  MoveL 1910 to (-109.13, -104.27, -4.96) mm, rotated rx 88.64 ry 0 rz 132.9 deg; joints [121.787, -25.073, 45.669, -119.581, 37.28, 191.868, 25, -132.901]
  MoveL 1911 to (-113.05, -99.53, -11.02) mm, rotated rx 86.5 ry 0 rz 130.7 deg; joints [121.42, -25.047, 46.567, -120.984, 37.45, 195.607, 25, -130.697]
  MoveL 1912 to (-113.34, -99.15, -11.43) mm, rotated rx 86.38 ry 0 rz 130.56 deg; joints [121.402, -25.048, 46.621, -121.062, 37.463, 195.813, 25, -130.561]
  MoveL 1913 to (-115.31, -96.51, -13.99) mm, rotated rx 85.43 ry 0 rz 129.34 deg; joints [121.25, -25.013, 47.005, -121.68, 37.561, 197.469, 25, -129.342]
  MoveL 1914 to (-115.68, -96.01, -14.39) mm, rotated rx 85.34 ry 0 rz 129.19 deg; joints [121.239, -25.019, 47.054, -121.738, 37.575, 197.627, 25, -129.193]
  MoveL 1915 to (-118.09, -92.7, -16.37) mm, rotated rx 84.63 ry 0 rz 127.72 deg; joints [121.132, -24.991, 47.345, -122.198, 37.66, 198.867, 25, -127.716]
  MoveL 1916 to (-118.46, -92.16, -16.77) mm, rotated rx 84.44 ry 0 rz 127.39 deg; joints [121.1, -24.97, 47.412, -122.327, 37.681, 199.21, 25, -127.39]
  MoveL 1917 to (-121.85, -86.42, -22.18) mm, rotated rx 82.29 ry 0 rz 124.74 deg; joints [120.788, -24.794, 48.227, -123.721, 37.981, 202.967, 25, -124.738]
  MoveL 1918 to (-122.46, -84.98, -24.25) mm, rotated rx 81.33 ry 0 rz 123.99 deg; joints [120.657, -24.684, 48.564, -124.332, 38.131, 204.635, 25, -123.992]
  MoveL 1919 to (-122.65, -84.59, -24.68) mm, rotated rx 81.33 ry 0 rz 123.99 deg; joints [120.661, -24.702, 48.591, -124.337, 38.14, 204.644, 25, -123.992]
  MoveL 1920 to (-122.81, -84.27, -24.97) mm, rotated rx 81.22 ry 0 rz 123.85 deg; joints [120.647, -24.69, 48.632, -124.407, 38.159, 204.837, 25, -123.853]
  MoveL 1921 to (-124.4, -81.2, -27.15) mm, rotated rx 80.44 ry 0 rz 122.62 deg; joints [120.554, -24.613, 48.934, -124.902, 38.304, 206.195, 25, -122.615]
  MoveL 1922 to (-124.78, -79.6, -30.03) mm, rotated rx 78.99 ry 0 rz 121.69 deg; joints [120.374, -24.397, 49.413, -125.811, 38.573, 208.715, 25, -121.69]
  MoveL 1923 to (-124.89, -79.17, -30.67) mm, rotated rx 78.81 ry 0 rz 121.57 deg; joints [120.355, -24.376, 49.486, -125.927, 38.614, 209.031, 25, -121.568]
  MoveL 1924 to (-125.14, -77.59, -33.5) mm, rotated rx 77.62 ry 0 rz 120.94 deg; joints [120.228, -24.195, 49.899, -126.663, 38.874, 211.098, 25, -120.935]
  MoveL 1925 to (-125.14, -77.57, -33.6) mm, rotated rx 76.62 ry 0 rz 120.98 deg; joints [120.153, -24.074, 50.182, -127.145, 39.063, 212.676, 25, -120.981]
  MoveL 1926 to (-124.65, -77.98, -34.49) mm, rotated rx 76.27 ry 0 rz 121.22 deg; joints [120.121, -24.015, 50.302, -127.356, 39.148, 213.273, 25, -121.217]
  MoveL 1927 to (-124.35, -78.16, -35.13) mm, rotated rx 76.27 ry 0 rz 121.22 deg; joints [120.109, -23.99, 50.31, -127.401, 39.159, 213.325, 25, -121.217]
  MoveL 1928 to (-124.19, -78.22, -35.56) mm, rotated rx 76.11 ry 0 rz 121.27 deg; joints [120.094, -23.961, 50.368, -127.503, 39.201, 213.615, 25, -121.269]
  MoveL 1929 to (-123.95, -78.19, -36.45) mm, rotated rx 76.11 ry 0 rz 121.27 deg; joints [120.085, -23.943, 50.39, -127.552, 39.22, 213.673, 25, -121.269]
  MoveL 1930 to (-123.38, -77.54, -39.6) mm, rotated rx 74.87 ry 0 rz 121.17 deg; joints [119.981, -23.712, 50.808, -128.292, 39.545, 215.805, 25, -121.168]
  MoveL 1931 to (-120.74, -79.41, -43.84) mm, rotated rx 72.6 ry 0 rz 122.5 deg; joints [119.836, -23.279, 51.521, -129.525, 40.165, 219.593, 25, -122.503]
  MoveL 1932 to (-120.21, -79.55, -45.03) mm, rotated rx 72.6 ry 0 rz 122.5 deg; joints [119.821, -23.236, 51.54, -129.599, 40.194, 219.681, 25, -122.503]
  MoveL 1933 to (-119.97, -79.45, -45.84) mm, rotated rx 72.28 ry 0 rz 122.52 deg; joints [119.801, -23.161, 51.642, -129.781, 40.294, 220.231, 25, -122.52]
  MoveL 1934 to (-117.99, -78.14, -52.73) mm, rotated rx 69.57 ry 0 rz 122.5 deg; joints [119.669, -22.465, 52.47, -131.278, 41.197, 224.832, 25, -122.503]
  MoveL 1935 to (-116.68, -77.5, -56.45) mm, rotated rx 68.02 ry 0 rz 122.57 deg; joints [119.621, -22.022, 52.911, -132.08, 41.754, 227.415, 25, -122.572]
  MoveL 1936 to (-116.44, -76.93, -57.7) mm, rotated rx 68.02 ry 0 rz 122.57 deg; joints [119.626, -22.007, 52.954, -132.122, 41.795, 227.475, 25, -122.572]
  MoveL 1937 to (-116.45, -76.65, -58.07) mm, rotated rx 67.87 ry 0 rz 122.47 deg; joints [119.622, -21.962, 52.996, -132.199, 41.852, 227.727, 25, -122.474]
  MoveL 1938 to (-116.52, -76.14, -58.6) mm, rotated rx 67.87 ry 0 rz 122.47 deg; joints [119.631, -21.972, 53.025, -132.204, 41.871, 227.74, 25, -122.474]
  MoveL 1939 to (-117.45, -71.82, -62.09) mm, rotated rx 66.42 ry 0 rz 120.74 deg; joints [119.607, -21.514, 53.417, -132.923, 42.43, 230.138, 25, -120.743]
  MoveL 1940 to (-117.61, -71.24, -62.45) mm, rotated rx 66.42 ry 0 rz 120.74 deg; joints [119.62, -21.534, 53.445, -132.916, 42.444, 230.138, 25, -120.743]
  MoveL 1941 to (-117.78, -70.77, -62.67) mm, rotated rx 66.33 ry 0 rz 120.54 deg; joints [119.619, -21.504, 53.469, -132.96, 42.48, 230.287, 25, -120.541]
  MoveL 1942 to (-119.62, -65.95, -64.4) mm, rotated rx 65.65 ry 0 rz 118.51 deg; joints [119.619, -21.283, 53.659, -133.285, 42.761, 231.416, 25, -118.506]
  MoveL 1943 to (-119.93, -63.2, -66.55) mm, rotated rx 64.56 ry 0 rz 117.09 deg; joints [119.603, -20.877, 53.896, -133.804, 43.193, 233.202, 25, -117.086]
  MoveL 1944 to (-120.07, -62.36, -67.09) mm, rotated rx 64.4 ry 0 rz 116.84 deg; joints [119.609, -20.828, 53.946, -133.874, 43.266, 233.458, 25, -116.837]
  MoveL 1945 to (-120.27, -59.5, -69.25) mm, rotated rx 63.41 ry 0 rz 115.6 deg; joints [119.614, -20.455, 54.174, -134.322, 43.687, 235.077, 25, -115.604]
  MoveL 1946 to (-120.29, -59.56, -69.2) mm, rotated rx 62.39 ry 0 rz 115.34 deg; joints [119.613, -20.12, 54.335, -134.692, 44.035, 236.603, 25, -115.342]
  MoveL 1947 to (-119.61, -59.72, -70.24) mm, rotated rx 61.95 ry 0 rz 115.53 deg; joints [119.623, -19.948, 54.435, -134.879, 44.231, 237.311, 25, -115.527]
  MoveL 1948 to (-119.15, -59.77, -70.98) mm, rotated rx 61.71 ry 0 rz 115.61 deg; joints [119.628, -19.842, 54.491, -134.99, 44.349, 237.717, 25, -115.606]
  MoveL 1949 to (-118.82, -59.72, -71.58) mm, rotated rx 61.71 ry 0 rz 115.61 deg; joints [119.628, -19.815, 54.5, -135.017, 44.374, 237.754, 25, -115.606]
  MoveL 1950 to (-115.87, -58.28, -77.36) mm, rotated rx 59.18 ry 0 rz 115.6 deg; joints [119.722, -18.764, 55.025, -136.014, 45.553, 241.762, 25, -115.596]
  MoveL 1951 to (-115.4, -57.54, -78.6) mm, rotated rx 59.18 ry 0 rz 115.6 deg; joints [119.738, -18.736, 55.064, -136.041, 45.61, 241.814, 25, -115.596]
  MoveL 1952 to (-115.3, -56.99, -79.15) mm, rotated rx 58.94 ry 0 rz 115.39 deg; joints [119.75, -18.628, 55.111, -136.132, 45.728, 242.2, 25, -115.393]
  MoveL 1953 to (-115.31, -56.09, -79.78) mm, rotated rx 58.94 ry 0 rz 115.39 deg; joints [119.771, -18.644, 55.152, -136.125, 45.758, 242.208, 25, -115.393]
  MoveL 1954 to (-116.04, -50.67, -82.28) mm, rotated rx 57.81 ry 0 rz 113.03 deg; joints [119.834, -18.134, 55.361, -136.531, 46.313, 243.977, 25, -113.033]
  MoveL 1955 to (-115.37, -50.42, -83.39) mm, rotated rx 56.63 ry 0 rz 112.48 deg; joints [119.873, -17.588, 55.497, -136.927, 46.83, 245.769, 25, -112.482]
  MoveL 1956 to (-115.05, -50.09, -84.03) mm, rotated rx 56.53 ry 0 rz 112.46 deg; joints [119.886, -17.528, 55.525, -136.969, 46.902, 245.943, 25, -112.463]
  MoveL 1957 to (-113.62, -47.98, -87.15) mm, rotated rx 55.08 ry 0 rz 111.8 deg; joints [119.994, -16.827, 55.753, -137.427, 47.641, 248.16, 25, -111.804]
  MoveL 1958 to (-113.36, -47.37, -87.82) mm, rotated rx 54.96 ry 0 rz 111.7 deg; joints [120.013, -16.758, 55.787, -137.469, 47.728, 248.366, 25, -111.704]
  MoveL 1959 to (-113.25, -46.78, -88.28) mm, rotated rx 54.96 ry 0 rz 111.7 deg; joints [120.028, -16.76, 55.812, -137.466, 47.752, 248.375, 25, -111.704]
  MoveL 1960 to (-113, -43.69, -90.16) mm, rotated rx 54.07 ry 0 rz 110.38 deg; joints [120.104, -16.312, 55.939, -137.728, 48.216, 249.725, 25, -110.383]
  MoveL 1961 to (-111.7, -40.57, -93.19) mm, rotated rx 52.42 ry 0 rz 108.96 deg; joints [120.248, -15.45, 56.129, -138.184, 49.072, 252.205, 25, -108.961]
  MoveL 1962 to (-111.45, -39.65, -93.88) mm, rotated rx 52.22 ry 0 rz 108.71 deg; joints [120.278, -15.34, 56.167, -138.235, 49.197, 252.516, 25, -108.714]
  MoveL 1963 to (-110.29, -33.42, -97.61) mm, rotated rx 50.45 ry 0 rz 106.05 deg; joints [120.479, -14.375, 56.365, -138.661, 50.167, 255.147, 25, -106.05]
  MoveL 1964 to (-110.16, -32.55, -98.04) mm, rotated rx 50.3 ry 0 rz 105.76 deg; joints [120.503, -14.292, 56.389, -138.692, 50.259, 255.374, 25, -105.76]
  MoveL 1965 to (-110.14, -31.93, -98.28) mm, rotated rx 50.3 ry 0 rz 105.76 deg; joints [120.519, -14.307, 56.413, -138.679, 50.274, 255.37, 25, -105.76]
  MoveL 1966 to (-110.3, -24.54, -100.19) mm, rotated rx 49.33 ry 0 rz 102.12 deg; joints [120.637, -13.76, 56.5, -138.888, 50.808, 256.791, 25, -102.124]
  MoveL 1967 to (-110.37, -23.8, -100.3) mm, rotated rx 49.33 ry 0 rz 102.12 deg; joints [120.655, -13.789, 56.528, -138.868, 50.816, 256.777, 25, -102.124]
  MoveL 1968 to (-110.46, -23.32, -100.31) mm, rotated rx 49.33 ry 0 rz 101.88 deg; joints [120.656, -13.785, 56.528, -138.869, 50.819, 256.788, 25, -101.875]
  MoveL 1969 to (-111.37, -19.04, -100.2) mm, rotated rx 49.38 ry 0 rz 99.74 deg; joints [120.653, -13.825, 56.53, -138.852, 50.789, 256.703, 25, -99.744]
  MoveL 1970 to (-111.19, -17.5, -100.68) mm, rotated rx 49.07 ry 0 rz 98.47 deg; joints [120.668, -13.604, 56.517, -138.946, 50.954, 257.182, 25, -98.467]
  MoveL 1971 to (-111.18, -16.84, -100.81) mm, rotated rx 49.07 ry 0 rz 98.47 deg; joints [120.684, -13.627, 56.542, -138.929, 50.963, 257.172, 25, -98.467]
  MoveL 1972 to (-111.39, -15.31, -100.82) mm, rotated rx 49.07 ry 0 rz 97.84 deg; joints [120.692, -13.641, 56.554, -138.92, 50.965, 257.166, 25, -97.845]
  MoveL 1973 to (-111.16, -13.52, -101.33) mm, rotated rx 48.75 ry 0 rz 96.5 deg; joints [120.712, -13.422, 56.546, -139.009, 51.133, 257.649, 25, -96.503]
  MoveL 1974 to (-111.2, -12.35, -101.43) mm, rotated rx 48.75 ry 0 rz 96.5 deg; joints [120.739, -13.472, 56.59, -138.975, 51.142, 257.624, 25, -96.503]
  MoveL 1975 to (-111.31, -11.84, -101.38) mm, rotated rx 48.77 ry 0 rz 96.23 deg; joints [120.736, -13.487, 56.588, -138.97, 51.127, 257.586, 25, -96.234]
  MoveL 1976 to (-112.07, -10.29, -100.7) mm, rotated rx 48.77 ry 0 rz 96.23 deg; joints [120.762, -13.607, 56.642, -138.905, 51.091, 257.512, 25, -96.234]
  MoveL 1977 to (-115.12, -7.08, -97.49) mm, rotated rx 50.4 ry 0 rz 94.47 deg; joints [120.561, -14.529, 56.499, -138.556, 50.192, 255.124, 25, -94.472]
  MoveL 1978 to (-116.27, -6.59, -96.15) mm, rotated rx 50.4 ry 0 rz 94.47 deg; joints [120.557, -14.636, 56.506, -138.505, 50.115, 255.041, 25, -94.472]
  MoveL 1979 to (-116.81, -6.76, -95.49) mm, rotated rx 50.49 ry 0 rz 94.48 deg; joints [120.538, -14.711, 56.487, -138.476, 50.036, 254.88, 25, -94.479]
  MoveL 1980 to (-117.52, -7.19, -94.57) mm, rotated rx 50.93 ry 0 rz 94.66 deg; joints [120.487, -14.956, 56.442, -138.37, 49.793, 254.222, 25, -94.66]
  MoveL 1981 to (-117.57, -7.2, -94.5) mm, rotated rx 51.73 ry 0 rz 94.56 deg; joints [120.413, -15.291, 56.364, -138.221, 49.448, 253.122, 25, -94.56]
  MoveL 1982 to (-119.21, -5.88, -92.53) mm, rotated rx 52.69 ry 0 rz 93.86 deg; joints [120.313, -15.805, 56.251, -137.973, 48.93, 251.683, 25, -93.861]
  MoveL 1983 to (-119.61, -5.59, -92.04) mm, rotated rx 52.87 ry 0 rz 93.75 deg; joints [120.296, -15.911, 56.229, -137.919, 48.827, 251.403, 25, -93.749]
  MoveL 1984 to (-122.12, -3.99, -88.75) mm, rotated rx 54.38 ry 0 rz 92.95 deg; joints [120.156, -16.699, 56.027, -137.487, 48.022, 249.109, 25, -92.949]
  MoveL 1985 to (-123.65, -1.68, -86.68) mm, rotated rx 55.61 ry 0 rz 91.63 deg; joints [120.049, -17.265, 55.833, -137.142, 47.407, 247.257, 25, -91.629]
  MoveL 1986 to (-124.31, -0.98, -85.75) mm, rotated rx 55.86 ry 0 rz 91.46 deg; joints [120.034, -17.423, 55.8, -137.039, 47.259, 246.842, 25, -91.458]
  MoveL 1987 to (-124.69, -0.74, -85.2) mm, rotated rx 55.86 ry 0 rz 91.46 deg; joints [120.036, -17.462, 55.801, -137.013, 47.232, 246.805, 25, -91.458]
  MoveL 1988 to (-128.3, 0.76, -79.65) mm, rotated rx 58.38 ry 0 rz 90.75 deg; joints [119.873, -18.639, 55.363, -136.152, 45.97, 242.887, 25, -90.746]
  MoveL 1989 to (-129.64, 1.6, -77.44) mm, rotated rx 59.45 ry 0 rz 90.34 deg; joints [119.818, -19.098, 55.159, -135.765, 45.463, 241.222, 25, -90.339]
  MoveL 1990 to (-130.13, 1.75, -76.61) mm, rotated rx 59.6 ry 0 rz 90.32 deg; joints [119.812, -19.188, 55.125, -135.686, 45.371, 240.957, 25, -90.323]
  MoveL 1991 to (-131.58, 1.85, -74.08) mm, rotated rx 60.65 ry 0 rz 90.28 deg; joints [119.77, -19.639, 54.906, -135.268, 44.869, 239.274, 25, -90.282]
  MoveL 1992 to (-131.68, 2.01, -73.92) mm, rotated rx 61.25 ry 0 rz 90 deg; joints [119.743, -19.816, 54.784, -135.087, 44.642, 238.395, 25, -90]
  MoveL 1993 to (-132.47, 3.26, -72.44) mm, rotated rx 61.9 ry 0 rz 89.46 deg; joints [119.724, -20.074, 54.643, -134.821, 44.348, 237.364, 25, -89.46]
  MoveL 1994 to (-132.84, 3.74, -71.74) mm, rotated rx 62.11 ry 0 rz 89.32 deg; joints [119.721, -20.174, 54.596, -134.718, 44.244, 237.004, 25, -89.32]
  MoveL 1995 to (-135.12, 6.38, -67.14) mm, rotated rx 64.03 ry 0 rz 88.24 deg; joints [119.691, -20.906, 54.148, -133.873, 43.401, 233.893, 25, -88.242]
  MoveL 1996 to (-136.66, 9.17, -63.61) mm, rotated rx 65.62 ry 0 rz 87.02 deg; joints [119.683, -21.451, 53.747, -133.148, 42.745, 231.299, 25, -87.023]
  MoveL 1997 to (-137.15, 9.63, -62.48) mm, rotated rx 65.62 ry 0 rz 87.02 deg; joints [119.693, -21.507, 53.736, -133.083, 42.705, 231.218, 25, -87.023]
  MoveL 1998 to (-137.46, 9.66, -61.8) mm, rotated rx 65.75 ry 0 rz 87.01 deg; joints [119.694, -21.56, 53.694, -133.007, 42.641, 230.989, 25, -87.014]
  MoveL 1999 to (-138.91, 9.39, -58.5) mm, rotated rx 67.12 ry 0 rz 87.16 deg; joints [119.71, -22.003, 53.33, -132.337, 42.104, 228.729, 25, -87.158]
  MoveL 2000 to (-139.18, 9.27, -57.89) mm, rotated rx 67.23 ry 0 rz 87.19 deg; joints [119.711, -22.044, 53.289, -132.27, 42.05, 228.528, 25, -87.188]
  MoveL 2001 to (-140.3, 7.99, -55.3) mm, rotated rx 68.09 ry 0 rz 87.65 deg; joints [119.728, -22.311, 53.03, -131.815, 41.709, 227.062, 25, -87.654]
  MoveL 2002 to (-140.85, 7.99, -53.9) mm, rotated rx 69.03 ry 0 rz 87.77 deg; joints [119.759, -22.574, 52.793, -131.357, 41.396, 225.532, 25, -87.767]
  MoveL 2003 to (-141.12, 7.84, -53.2) mm, rotated rx 69.03 ry 0 rz 87.77 deg; joints [119.757, -22.583, 52.77, -131.331, 41.374, 225.497, 25, -87.767]
  MoveL 2004 to (-141.46, 7.5, -52.35) mm, rotated rx 69.38 ry 0 rz 87.91 deg; joints [119.77, -22.68, 52.669, -131.149, 41.252, 224.918, 25, -87.908]
  MoveL 2005 to (-143.81, 3.71, -45.92) mm, rotated rx 71.82 ry 0 rz 89.38 deg; joints [119.882, -23.311, 51.913, -129.798, 40.426, 220.758, 25, -89.385]
  MoveL 2006 to (-143.79, 3.76, -45.99) mm, rotated rx 72.66 ry 0 rz 89.41 deg; joints [119.923, -23.469, 51.711, -129.425, 40.224, 219.457, 25, -89.408]
  MoveL 2007 to (-144.66, 5.18, -43.07) mm, rotated rx 73.82 ry 0 rz 88.85 deg; joints [120, -23.726, 51.335, -128.753, 39.878, 217.462, 25, -88.851]
  MoveL 2008 to (-144.92, 5.41, -42.15) mm, rotated rx 73.82 ry 0 rz 88.85 deg; joints [120.011, -23.754, 51.317, -128.699, 39.857, 217.398, 25, -88.851]
  MoveL 2009 to (-145.17, 5.36, -41.27) mm, rotated rx 73.92 ry 0 rz 88.85 deg; joints [120.02, -23.783, 51.266, -128.613, 39.813, 217.193, 25, -88.847]
  MoveL 2010 to (-145.6, 4.99, -39.76) mm, rotated rx 75.16 ry 0 rz 88.92 deg; joints [120.101, -23.992, 50.893, -127.972, 39.509, 215.173, 25, -88.915]
  MoveL 2011 to (-146.32, 6.55, -36.79) mm, rotated rx 76.33 ry 0 rz 88.31 deg; joints [120.202, -24.206, 50.495, -127.268, 39.207, 213.153, 25, -88.309]
  MoveL 2012 to (-146.5, 7.02, -35.98) mm, rotated rx 76.68 ry 0 rz 88.11 deg; joints [120.233, -24.263, 50.375, -127.062, 39.122, 212.555, 25, -88.11]
  MoveL 2013 to (-147.72, 11.76, -29.12) mm, rotated rx 79.41 ry 0 rz 86.25 deg; joints [120.514, -24.663, 49.403, -125.378, 38.516, 207.815, 25, -86.25]
  MoveL 2014 to (-147.89, 15.71, -26.25) mm, rotated rx 80.75 ry 0 rz 84.52 deg; joints [120.655, -24.79, 48.909, -124.585, 38.265, 205.54, 25, -84.518]
  MoveL 2015 to (-147.93, 16.33, -25.65) mm, rotated rx 80.87 ry 0 rz 84.41 deg; joints [120.68, -24.822, 48.867, -124.48, 38.242, 205.302, 25, -84.407]
  MoveL 2016 to (-148.25, 18.54, -22.05) mm, rotated rx 82.08 ry 0 rz 83.7 deg; joints [120.85, -24.964, 48.406, -123.666, 38.034, 203.142, 25, -83.704]
  MoveL 2017 to (-148.41, 18.88, -20.63) mm, rotated rx 82.08 ry 0 rz 83.7 deg; joints [120.873, -24.99, 48.373, -123.578, 38.018, 203.042, 25, -83.704]
  MoveL 2018 to (-148.62, 18.58, -19.38) mm, rotated rx 82.16 ry 0 rz 83.71 deg; joints [120.889, -24.99, 48.297, -123.48, 37.989, 202.838, 25, -83.71]
  MoveL 2019 to (-148.94, 17.65, -17.69) mm, rotated rx 82.81 ry 0 rz 84.07 deg; joints [120.979, -25.044, 48.049, -123.063, 37.892, 201.707, 25, -84.074]
  MoveL 2020 to (-149.44, 16.99, -13.68) mm, rotated rx 84.63 ry 0 rz 84.45 deg; joints [121.245, -25.175, 47.37, -121.909, 37.664, 198.556, 25, -84.448]
  MoveL 2021 to (-149.51, 16.81, -13.05) mm, rotated rx 84.73 ry 0 rz 84.48 deg; joints [121.263, -25.177, 47.317, -121.83, 37.649, 198.368, 25, -84.483]
  MoveL 2022 to (-149.73, 16.26, -10.96) mm, rotated rx 85.58 ry 0 rz 84.72 deg; joints [121.397, -25.219, 46.983, -121.28, 37.558, 196.882, 25, -84.72]
  MoveL 2023 to (-149.72, 16.22, -11.05) mm, rotated rx 86.54 ry 0 rz 84.42 deg; joints [121.5, -25.207, 46.658, -120.829, 37.479, 195.406, 25, -84.417]
  MoveL 2024 to (-149.59, 18.71, -8.96) mm, rotated rx 87.54 ry 0 rz 83 deg; joints [121.633, -25.173, 46.232, -120.256, 37.386, 193.745, 25, -82.996]
  MoveL 2025 to (-148.52, 25.7, -9.48) mm, rotated rx 87.35 ry 0 rz 80.12 deg; joints [121.588, -25.145, 46.294, -120.402, 37.396, 194.1, 25, -80.117]
  MoveL 2026 to (-148.27, 27.19, -9.1) mm, rotated rx 87.35 ry 0 rz 80.12 deg; joints [121.628, -25.218, 46.329, -120.32, 37.409, 194.015, 25, -80.117]
  MoveL 2027 to (-148.17, 27.92, -8.63) mm, rotated rx 87.52 ry 0 rz 79.84 deg; joints [121.658, -25.221, 46.257, -120.205, 37.395, 193.707, 25, -79.837]
  MoveL 2028 to (-147.29, 33.08, -4.1) mm, rotated rx 89.39 ry 0 rz 77.41 deg; joints [121.959, -25.182, 45.465, -119.059, 37.268, 190.534, 25, -77.412]
  MoveL 2029 to (-147.14, 33.77, -4.05) mm, rotated rx 89.41 ry 0 rz 77.15 deg; joints [121.963, -25.182, 45.457, -119.046, 37.267, 190.499, 25, -77.146]
  MoveL 2030 to (-143.96, 45.19, -6.36) mm, rotated rx 88.52 ry 0 rz 72.4 deg; joints [121.787, -25.149, 45.804, -119.648, 37.309, 192.069, 25, -72.396]
  MoveL 2031 to (-142.1, 50.49, -8.11) mm, rotated rx 87.83 ry 0 rz 70.16 deg; joints [121.66, -25.128, 46.078, -120.106, 37.353, 193.28, 25, -70.162]
  MoveL 2032 to (-141.84, 51.2, -8.22) mm, rotated rx 87.83 ry 0 rz 70.16 deg; joints [121.676, -25.164, 46.105, -120.081, 37.361, 193.256, 25, -70.162]
  MoveL 2033 to (-141.67, 51.67, -8.22) mm, rotated rx 87.83 ry 0 rz 69.97 deg; joints [121.676, -25.163, 46.104, -120.081, 37.361, 193.254, 25, -69.968]
  MoveL 2034 to (-139.95, 56.28, -7.34) mm, rotated rx 88.15 ry 0 rz 68.27 deg; joints [121.742, -25.189, 45.986, -119.854, 37.343, 192.681, 25, -68.267]
  MoveL 2035 to (-137.43, 62.13, -7.66) mm, rotated rx 88.04 ry 0 rz 65.63 deg; joints [121.709, -25.16, 46.013, -119.949, 37.345, 192.893, 25, -65.625]
  MoveL 2036 to (-135.16, 66.76, -9.11) mm, rotated rx 87.45 ry 0 rz 63.46 deg; joints [121.597, -25.123, 46.232, -120.348, 37.382, 193.929, 25, -63.458]
  MoveL 2037 to (-134.83, 67.4, -9.2) mm, rotated rx 87.45 ry 0 rz 63.46 deg; joints [121.612, -25.158, 46.258, -120.323, 37.39, 193.904, 25, -63.458]
  MoveL 2038 to (-134.37, 68.32, -9.18) mm, rotated rx 87.46 ry 0 rz 63.07 deg; joints [121.613, -25.158, 46.255, -120.318, 37.389, 193.891, 25, -63.066]
  MoveL 2039 to (-133.91, 69.25, -8.94) mm, rotated rx 87.46 ry 0 rz 63.07 deg; joints [121.64, -25.207, 46.278, -120.264, 37.398, 193.834, 25, -63.066]
  MoveL 2040 to (-130.27, 76.23, -5.17) mm, rotated rx 88.89 ry 0 rz 60.07 deg; joints [121.892, -25.224, 45.691, -119.333, 37.302, 191.347, 25, -60.072]
  MoveL 2041 to (-129.97, 76.76, -4.82) mm, rotated rx 88.98 ry 0 rz 59.92 deg; joints [121.915, -25.234, 45.656, -119.259, 37.299, 191.173, 25, -59.921]
  MoveL 2042 to (-128.21, 79.76, -2.85) mm, rotated rx 89.74 ry 0 rz 58.58 deg; joints [122.053, -25.229, 45.339, -118.771, 37.261, 189.86, 25, -58.583]
  MoveL 2043 to (-127.99, 80.12, -2.6) mm, rotated rx 89.83 ry 0 rz 58.43 deg; joints [122.071, -25.229, 45.302, -118.712, 37.258, 189.703, 25, -58.427]
  MoveL 2044 to (-126.08, 83.14, -0.8) mm, rotated rx 90.54 ry 0 rz 57.03 deg; joints [122.201, -25.214, 45.003, -118.261, 37.23, 188.483, 25, -57.026]
  MoveL 2045 to (-125.78, 83.59, -0.43) mm, rotated rx 90.54 ry 0 rz 57.03 deg; joints [122.22, -25.239, 45.007, -118.22, 37.235, 188.439, 25, -57.026]
  MoveL 2046 to (-125.56, 83.91, -0.09) mm, rotated rx 90.67 ry 0 rz 56.88 deg; joints [122.245, -25.237, 44.952, -118.136, 37.231, 188.214, 25, -56.881]
  MoveL 2047 to (-125.22, 84.42, 0.77) mm, rotated rx 90.67 ry 0 rz 56.88 deg; joints [122.272, -25.264, 44.941, -118.067, 37.236, 188.139, 25, -56.881]
  MoveL 2048 to (-124.21, 85.78, 4.61) mm, rotated rx 92.13 ry 0 rz 56.24 deg; joints [122.56, -25.221, 44.323, -117.134, 37.211, 185.631, 25, -56.242]
  MoveL 2049 to (-121.27, 89.62, 8.28) mm, rotated rx 93.9 ry 0 rz 54.11 deg; joints [122.892, -25.104, 43.573, -116.097, 37.208, 182.696, 25, -54.113]
  MoveL 2050 to (-120.98, 89.99, 8.63) mm, rotated rx 94.04 ry 0 rz 53.92 deg; joints [122.921, -25.094, 43.512, -116.012, 37.21, 182.459, 25, -53.921]
  MoveL 2051 to (-117.7, 93.74, 12.84) mm, rotated rx 95.6 ry 0 rz 52.08 deg; joints [123.265, -24.993, 42.831, -115.03, 37.255, 179.797, 25, -52.083]
  MoveL 2052 to (-117.06, 94.32, 14.38) mm, rotated rx 95.6 ry 0 rz 52.08 deg; joints [123.313, -25.022, 42.801, -114.921, 37.272, 179.679, 25, -52.083]
  MoveL 2053 to (-116.97, 94.28, 15.39) mm, rotated rx 95.69 ry 0 rz 52.07 deg; joints [123.347, -25.009, 42.734, -114.828, 37.278, 179.484, 25, -52.07]
  MoveL 2054 to (-117, 93.95, 17.04) mm, rotated rx 96.32 ry 0 rz 52.18 deg; joints [123.489, -24.956, 42.456, -114.442, 37.308, 178.422, 25, -52.177]
  MoveL 2055 to (-116.24, 94.53, 18.96) mm, rotated rx 97.62 ry 0 rz 51.74 deg; joints [123.755, -24.836, 41.927, -113.738, 37.373, 176.335, 25, -51.744]
  MoveL 2056 to (-115.96, 94.57, 20.45) mm, rotated rx 97.62 ry 0 rz 51.74 deg; joints [123.788, -24.833, 41.879, -113.658, 37.384, 176.246, 25, -51.744]
  MoveL 2057 to (-116.14, 94.01, 21.92) mm, rotated rx 97.76 ry 0 rz 51.77 deg; joints [123.83, -24.787, 41.763, -113.54, 37.392, 175.976, 25, -51.767]
  MoveL 2058 to (-117.02, 92.32, 24.27) mm, rotated rx 99.1 ry 0 rz 52.68 deg; joints [124.137, -24.671, 41.221, -112.789, 37.495, 173.806, 25, -52.677]
  MoveL 2059 to (-116.98, 92.03, 25.56) mm, rotated rx 99.59 ry 0 rz 52.76 deg; joints [124.257, -24.612, 40.999, -112.502, 37.538, 172.99, 25, -52.759]
  MoveL 2060 to (-117.05, 91.68, 26.5) mm, rotated rx 99.75 ry 0 rz 52.82 deg; joints [124.302, -24.581, 40.905, -112.392, 37.554, 172.712, 25, -52.823]
  MoveL 2061 to (-117.17, 90.63, 29.37) mm, rotated rx 100.93 ry 0 rz 53.2 deg; joints [124.592, -24.431, 40.379, -111.723, 37.671, 170.784, 25, -53.202]
  MoveL 2062 to (-116.45, 90.99, 31.12) mm, rotated rx 102.26 ry 0 rz 52.89 deg; joints [124.888, -24.259, 39.839, -111.065, 37.802, 168.732, 25, -52.894]
  MoveL 2063 to (-116.16, 91, 32.15) mm, rotated rx 102.26 ry 0 rz 52.89 deg; joints [124.914, -24.254, 39.806, -111.012, 37.816, 168.674, 25, -52.894]
  MoveL 2064 to (-116.09, 90.62, 33.43) mm, rotated rx 103.42 ry 0 rz 52.76 deg; joints [125.162, -24.071, 39.323, -110.478, 37.933, 166.921, 25, -52.755]
  MoveL 2065 to (-114.95, 91.49, 34.97) mm, rotated rx 104.01 ry 0 rz 52.22 deg; joints [125.317, -23.974, 39.05, -110.158, 38.012, 165.97, 25, -52.216]
  MoveL 2066 to (-114.26, 91.74, 36.56) mm, rotated rx 104.01 ry 0 rz 52.22 deg; joints [125.367, -23.979, 39.007, -110.068, 38.04, 165.871, 25, -52.216]
  MoveL 2067 to (-114.19, 91.07, 38.4) mm, rotated rx 104.17 ry 0 rz 52.22 deg; joints [125.428, -23.912, 38.865, -109.936, 38.071, 165.566, 25, -52.216]
  MoveL 2068 to (-115.08, 88.3, 42.05) mm, rotated rx 105.61 ry 0 rz 53.3 deg; joints [125.811, -23.66, 38.204, -109.191, 38.282, 163.302, 25, -53.302]
  MoveL 2069 to (-115.21, 87.18, 43.98) mm, rotated rx 106.52 ry 0 rz 53.78 deg; joints [126.052, -23.507, 37.806, -108.742, 38.424, 161.902, 25, -53.775]
  MoveL 2070 to (-115.3, 86.78, 44.52) mm, rotated rx 106.52 ry 0 rz 53.78 deg; joints [126.056, -23.482, 37.774, -108.731, 38.425, 161.889, 25, -53.775]
  MoveL 2071 to (-115.4, 86.48, 44.85) mm, rotated rx 106.64 ry 0 rz 53.9 deg; joints [126.091, -23.457, 37.715, -108.667, 38.446, 161.688, 25, -53.896]
  MoveL 2072 to (-116.47, 83.68, 47.31) mm, rotated rx 107.55 ry 0 rz 54.97 deg; joints [126.339, -23.269, 37.282, -108.22, 38.597, 160.289, 25, -54.966]
  MoveL 2073 to (-116.37, 82.67, 49.3) mm, rotated rx 108.7 ry 0 rz 55.54 deg; joints [126.651, -23.077, 36.803, -107.687, 38.797, 158.555, 25, -55.536]
  MoveL 2074 to (-116.42, 82.21, 49.94) mm, rotated rx 108.7 ry 0 rz 55.54 deg; joints [126.657, -23.048, 36.766, -107.674, 38.799, 158.539, 25, -55.536]
  MoveL 2075 to (-116.6, 81.61, 50.52) mm, rotated rx 108.79 ry 0 rz 55.62 deg; joints [126.681, -23.007, 36.698, -107.629, 38.814, 158.397, 25, -55.618]
  MoveL 2076 to (-117.58, 78.88, 52.54) mm, rotated rx 109.6 ry 0 rz 56.76 deg; joints [126.909, -22.833, 36.32, -107.251, 38.964, 157.167, 25, -56.756]
  MoveL 2077 to (-117.87, 77.18, 54.39) mm, rotated rx 110.51 ry 0 rz 57.57 deg; joints [127.166, -22.658, 35.926, -106.844, 39.139, 155.815, 25, -57.568]
  MoveL 2078 to (-118.08, 76.44, 54.96) mm, rotated rx 110.51 ry 0 rz 57.57 deg; joints [127.162, -22.617, 35.882, -106.843, 39.134, 155.813, 25, -57.568]
  MoveL 2079 to (-118.37, 75.77, 55.27) mm, rotated rx 110.56 ry 0 rz 57.67 deg; joints [127.17, -22.583, 35.837, -106.825, 39.139, 155.738, 25, -57.675]
  MoveL 2080 to (-119.55, 73.3, 56.05) mm, rotated rx 110.88 ry 0 rz 58.79 deg; joints [127.261, -22.51, 35.689, -106.683, 39.202, 155.263, 25, -58.787]
  MoveL 2081 to (-119.75, 72.81, 56.26) mm, rotated rx 110.99 ry 0 rz 59.09 deg; joints [127.297, -22.494, 35.645, -106.63, 39.227, 155.091, 25, -59.087]
  MoveL 2082 to (-120.75, 68.2, 59.75) mm, rotated rx 112.58 ry 0 rz 61.2 deg; joints [127.759, -22.155, 34.939, -105.943, 39.557, 152.754, 25, -61.2]
  MoveL 2083 to (-120.68, 68.16, 59.97) mm, rotated rx 113.09 ry 0 rz 61.52 deg; joints [127.902, -22.083, 34.761, -105.743, 39.662, 152.018, 25, -61.52]
  MoveL 2084 to (-119.88, 66.14, 63.73) mm, rotated rx 114.66 ry 0 rz 62.1 deg; joints [128.359, -21.69, 34.029, -105.11, 40.002, 149.755, 25, -62.103]
  MoveL 2085 to (-119.8, 65.76, 64.28) mm, rotated rx 114.66 ry 0 rz 62.1 deg; joints [128.366, -21.666, 33.998, -105.098, 40.006, 149.742, 25, -62.103]
  MoveL 2086 to (-119.77, 65.42, 64.66) mm, rotated rx 114.82 ry 0 rz 62.22 deg; joints [128.414, -21.624, 33.922, -105.034, 40.043, 149.508, 25, -62.225]
  MoveL 2087 to (-119.95, 61.76, 67.86) mm, rotated rx 116.05 ry 0 rz 63.53 deg; joints [128.776, -21.286, 33.331, -104.561, 40.32, 147.768, 25, -63.527]
  MoveL 2088 to (-120.08, 60.96, 68.35) mm, rotated rx 116.05 ry 0 rz 63.53 deg; joints [128.77, -21.245, 33.289, -104.564, 40.315, 147.77, 25, -63.527]
  MoveL 2089 to (-120.24, 60.38, 68.59) mm, rotated rx 116.15 ry 0 rz 63.78 deg; joints [128.801, -21.217, 33.241, -104.525, 40.339, 147.623, 25, -63.78]
  MoveL 2090 to (-120.98, 56.47, 70.56) mm, rotated rx 117.04 ry 0 rz 65.51 deg; joints [129.067, -20.986, 32.836, -104.196, 40.548, 146.377, 25, -65.512]
  MoveL 2091 to (-118.84, 57.87, 73.02) mm, rotated rx 119.86 ry 0 rz 64.15 deg; joints [129.775, -20.257, 31.666, -103.367, 41.117, 142.647, 25, -64.146]
  MoveL 2092 to (-117.93, 59.53, 73.19) mm, rotated rx 119.93 ry 0 rz 63.32 deg; joints [129.797, -20.236, 31.632, -103.343, 41.134, 142.548, 25, -63.323]
  MoveL 2093 to (-116.76, 60.86, 73.96) mm, rotated rx 119.96 ry 0 rz 63.31 deg; joints [129.867, -20.272, 31.633, -103.273, 41.193, 142.445, 25, -63.31]
  MoveL 2094 to (-115.68, 60.98, 75.54) mm, rotated rx 119.99 ry 0 rz 63.3 deg; joints [129.932, -20.243, 31.57, -103.204, 41.247, 142.342, 25, -63.297]
  MoveL 2095 to (-115.1, 60.65, 76.68) mm, rotated rx 120.49 ry 0 rz 63.32 deg; joints [130.083, -20.095, 31.336, -103.041, 41.372, 141.664, 25, -63.315]
  MoveL 2096 to (-114.03, 60.99, 78.01) mm, rotated rx 121.53 ry 0 rz 62.85 deg; joints [130.362, -19.803, 30.89, -102.749, 41.604, 140.307, 25, -62.85]
  MoveL 2097 to (-113.32, 60.92, 79.08) mm, rotated rx 121.53 ry 0 rz 62.85 deg; joints [130.399, -19.782, 30.85, -102.712, 41.636, 140.267, 25, -62.85]
  MoveL 2098 to (-112.82, 60.37, 80.21) mm, rotated rx 121.68 ry 0 rz 62.86 deg; joints [130.462, -19.704, 30.738, -102.647, 41.688, 140.045, 25, -62.86]
  MoveL 2099 to (-111.85, 57.98, 83.26) mm, rotated rx 123.17 ry 0 rz 63.58 deg; joints [130.904, -19.247, 30.054, -102.212, 42.063, 138.085, 25, -63.576]
  MoveL 2100 to (-109.17, 56.99, 87.4) mm, rotated rx 125.32 ry 0 rz 63.47 deg; joints [131.544, -18.579, 29.084, -101.628, 42.616, 135.306, 25, -63.472]
  MoveL 2101 to (-108.53, 56, 88.83) mm, rotated rx 125.32 ry 0 rz 63.47 deg; joints [131.572, -18.511, 29.003, -101.602, 42.641, 135.278, 25, -63.472]
  MoveL 2102 to (-108.42, 55.2, 89.47) mm, rotated rx 125.62 ry 0 rz 63.79 deg; joints [131.666, -18.411, 28.861, -101.521, 42.723, 134.883, 25, -63.795]
  MoveL 2103 to (-108.75, 53.37, 90.18) mm, rotated rx 125.62 ry 0 rz 63.79 deg; joints [131.642, -18.323, 28.781, -101.537, 42.702, 134.899, 25, -63.795]
  MoveL 2104 to (-112.59, 43.93, 90.56) mm, rotated rx 125.9 ry 0 rz 68.74 deg; joints [131.725, -18.25, 28.671, -101.467, 42.774, 134.553, 25, -68.74]
  MoveL 2105 to (-113.25, 41.96, 90.66) mm, rotated rx 125.95 ry 0 rz 69.76 deg; joints [131.743, -18.235, 28.649, -101.452, 42.79, 134.484, 25, -69.757]
  MoveL 2106 to (-113.56, 41.16, 90.65) mm, rotated rx 125.94 ry 0 rz 70.02 deg; joints [131.732, -18.227, 28.646, -101.46, 42.781, 134.503, 25, -70.02]
  MoveL 2107 to (-113.92, 38.56, 91.31) mm, rotated rx 126.3 ry 0 rz 71.64 deg; joints [131.861, -18.14, 28.506, -101.355, 42.894, 134.03, 25, -71.637]
  MoveL 2108 to (-113.89, 38.54, 91.36) mm, rotated rx 127.16 ry 0 rz 72.49 deg; joints [132.115, -17.973, 28.237, -101.149, 43.119, 132.946, 25, -72.494]
  MoveL 2109 to (-112.68, 37.99, 93.08) mm, rotated rx 128.64 ry 0 rz 72.32 deg; joints [132.509, -17.5, 27.608, -100.839, 43.471, 131.138, 25, -72.316]
  MoveL 2110 to (-110.38, 39.47, 95.21) mm, rotated rx 129.67 ry 0 rz 71.29 deg; joints [132.821, -17.145, 27.139, -100.607, 43.751, 129.866, 25, -71.29]
  MoveL 2111 to (-108.12, 42.41, 96.54) mm, rotated rx 130.58 ry 0 rz 69.14 deg; joints [133.06, -16.816, 26.726, -100.435, 43.967, 128.773, 25, -69.145]
  Set speed (16.7 mm/s)
  MoveL 2112 to (-122.31, 47.82, 109.55) mm, rotated rx 130.58 ry 0 rz 69.14 deg; joints [132.836, -17.119, 26.307, -99.772, 43.624, 127.803, 25, -69.145]
  Set speed (1000.0 mm/s)
  MoveL 2113 to (-119.4, 45.41, 113.71) mm, rotated rx 130.84 ry 0 rz 69.27 deg; joints [133.011, -16.856, 25.988, -99.655, 43.784, 127.419, 25, -69.275]
  Set speed (5.0 mm/s)
  MoveL 2114 to (-105.24, 40.05, 100.63) mm, rotated rx 130.84 ry 0 rz 69.27 deg; joints [133.231, -16.556, 26.409, -100.316, 44.123, 128.388, 25, -69.275]
  Set speed (16.7 mm/s)
  MoveL 2115 to (-106.36, 36.25, 100.88) mm, rotated rx 130.97 ry 0 rz 71.29 deg; joints [133.271, -16.51, 26.35, -100.29, 44.159, 128.232, 25, -71.288]
  Set speed (16.7 mm/s)
  MoveL 2116 to (-120.67, 41.09, 113.99) mm, rotated rx 130.97 ry 0 rz 71.29 deg; joints [133.052, -16.808, 25.928, -99.629, 43.822, 127.263, 25, -71.288]
  Set speed (1000.0 mm/s)
  MoveL 2117 to (-118.91, 26.12, 120.09) mm, rotated rx 134.04 ry 0 rz 78.48 deg; joints [134.034, -15.736, 24.575, -99.03, 44.733, 123.566, 25, -78.475]
  Set speed (5.0 mm/s)
  MoveL 2118 to (-104.82, 23.25, 106.19) mm, rotated rx 134.04 ry 0 rz 78.48 deg; joints [134.22, -15.471, 25.034, -99.688, 45.032, 124.537, 25, -78.475]
  Set speed (16.7 mm/s)
  MoveL 2119 to (-104.41, 21.99, 106.87) mm, rotated rx 134.42 ry 0 rz 79.11 deg; joints [134.332, -15.335, 24.869, -99.623, 45.136, 124.098, 25, -79.109]
  MoveL 2120 to (-102.69, 19.1, 109.07) mm, rotated rx 135.76 ry 0 rz 80.71 deg; joints [134.734, -14.857, 24.294, -99.397, 45.511, 122.53, 25, -80.706]
  MoveL 2121 to (-102.33, 17.43, 109.68) mm, rotated rx 135.76 ry 0 rz 80.71 deg; joints [134.715, -14.777, 24.22, -99.409, 45.494, 122.542, 25, -80.706]
  MoveL 2122 to (-102.37, 16.88, 109.73) mm, rotated rx 135.79 ry 0 rz 81.02 deg; joints [134.724, -14.767, 24.208, -99.404, 45.502, 122.509, 25, -81.016]
  MoveL 2123 to (-102.11, 14.05, 110.35) mm, rotated rx 136.17 ry 0 rz 82.81 deg; joints [134.849, -14.64, 24.053, -99.337, 45.619, 122.056, 25, -82.813]
  MoveL 2124 to (-102.17, 14.13, 110.3) mm, rotated rx 137.24 ry 0 rz 83.75 deg; joints [135.141, -14.38, 23.73, -99.184, 45.893, 120.841, 25, -83.753]
  MoveL 2125 to (-99.55, 14.42, 112.66) mm, rotated rx 138.55 ry 0 rz 83.46 deg; joints [135.531, -13.875, 23.151, -98.992, 46.262, 119.34, 25, -83.459]
  MoveL 2126 to (-97.81, 15.28, 114.06) mm, rotated rx 139.93 ry 0 rz 82.37 deg; joints [135.878, -13.36, 22.581, -98.834, 46.592, 117.817, 25, -82.375]
  MoveL 2127 to (-95.33, 17.87, 115.77) mm, rotated rx 140.85 ry 0 rz 80.73 deg; joints [136.155, -12.993, 22.175, -98.713, 46.856, 116.783, 25, -80.727]
  MoveL 2128 to (-94.23, 18.44, 116.58) mm, rotated rx 140.85 ry 0 rz 80.73 deg; joints [136.204, -12.976, 22.15, -98.691, 46.902, 116.762, 25, -80.727]
  MoveL 2129 to (-93.66, 18.46, 117.03) mm, rotated rx 140.94 ry 0 rz 80.7 deg; joints [136.242, -12.928, 22.097, -98.675, 46.939, 116.661, 25, -80.696]
  MoveL 2130 to (-92.1, 18.26, 118.3) mm, rotated rx 141.72 ry 0 rz 80.66 deg; joints [136.468, -12.618, 21.76, -98.584, 47.155, 115.797, 25, -80.664]
  MoveL 2131 to (-89.1, 18.17, 120.59) mm, rotated rx 143.24 ry 0 rz 80.4 deg; joints [136.898, -12.016, 21.116, -98.42, 47.569, 114.136, 25, -80.4]
  MoveL 2132 to (-88, 17.68, 121.46) mm, rotated rx 143.24 ry 0 rz 80.4 deg; joints [136.924, -11.959, 21.058, -98.411, 47.595, 114.129, 25, -80.4]
  MoveL 2133 to (-87.65, 17.34, 121.76) mm, rotated rx 143.43 ry 0 rz 80.58 deg; joints [136.98, -11.88, 20.975, -98.391, 47.649, 113.916, 25, -80.58]
  MoveL 2134 to (-87.09, 16.45, 122.28) mm, rotated rx 143.43 ry 0 rz 80.58 deg; joints [136.98, -11.827, 20.924, -98.393, 47.649, 113.92, 25, -80.58]
  MoveL 2135 to (-85.63, 12.54, 123.76) mm, rotated rx 144.42 ry 0 rz 83.04 deg; joints [137.264, -11.429, 20.508, -98.295, 47.923, 112.849, 25, -83.043]
  MoveL 2136 to (-84.87, 11.35, 124.41) mm, rotated rx 144.96 ry 0 rz 84.02 deg; joints [137.419, -11.23, 20.3, -98.242, 48.074, 112.269, 25, -84.018]
  MoveL 2137 to (-84.51, 10.45, 124.72) mm, rotated rx 144.96 ry 0 rz 84.02 deg; joints [137.41, -11.186, 20.259, -98.248, 48.065, 112.275, 25, -84.018]
  MoveL 2138 to (-84.4, 9.74, 124.85) mm, rotated rx 145.01 ry 0 rz 84.21 deg; joints [137.414, -11.151, 20.226, -98.248, 48.07, 112.233, 25, -84.214]
  MoveL 2139 to (-84.29, 8.18, 125.03) mm, rotated rx 145.13 ry 0 rz 85.28 deg; joints [137.449, -11.103, 20.176, -98.237, 48.104, 112.104, 25, -85.281]
  MoveL 2140 to (-84.32, 8.21, 125.03) mm, rotated rx 145.76 ry 0 rz 86.57 deg; joints [137.639, -10.957, 20.015, -98.17, 48.287, 111.413, 25, -86.567]
  MoveL 2141 to (-83.75, 7.93, 125.43) mm, rotated rx 146.04 ry 0 rz 86.74 deg; joints [137.716, -10.844, 19.901, -98.147, 48.362, 111.121, 25, -86.735]
  MoveL 2142 to (-83.33, 7.67, 125.72) mm, rotated rx 146.1 ry 0 rz 86.79 deg; joints [137.738, -10.801, 19.858, -98.141, 48.384, 111.054, 25, -86.795]
  MoveL 2143 to (-82.15, 6.44, 126.56) mm, rotated rx 146.53 ry 0 rz 87.43 deg; joints [137.861, -10.602, 19.658, -98.105, 48.504, 110.597, 25, -87.433]
  MoveL 2144 to (-81.38, 6.16, 127.08) mm, rotated rx 147.23 ry 0 rz 87.93 deg; joints [138.046, -10.359, 19.411, -98.05, 48.684, 109.866, 25, -87.929]
  MoveL 2145 to (-80.87, 5.85, 127.42) mm, rotated rx 147.23 ry 0 rz 87.93 deg; joints [138.053, -10.329, 19.382, -98.049, 48.691, 109.866, 25, -87.929]
  MoveL 2146 to (-80.53, 5.57, 127.65) mm, rotated rx 147.39 ry 0 rz 88.13 deg; joints [138.098, -10.261, 19.315, -98.037, 48.736, 109.693, 25, -88.125]
  MoveL 2147 to (-78.37, 3.33, 129.04) mm, rotated rx 148.32 ry 0 rz 89.61 deg; joints [138.355, -9.864, 18.922, -97.969, 48.988, 108.727, 25, -89.608]
  Set speed (16.7 mm/s)
  MoveL 2148 to (-88.88, 3.4, 146.06) mm, rotated rx 148.32 ry 0 rz 89.61 deg; joints [138.303, -9.967, 18.301, -97.358, 48.84, 107.784, 25, -89.608]
  Set speed (1000.0 mm/s)
  MoveL 2149 to (-85.2, 1.1, 148.27) mm, rotated rx 149.48 ry 0 rz 90 deg; joints [138.606, -9.387, 17.74, -97.297, 49.14, 106.595, 25, -90]
  Set speed (5.0 mm/s)
  MoveL 2150 to (-75.05, 1.1, 131.04) mm, rotated rx 149.48 ry 0 rz 90 deg; joints [138.649, -9.297, 18.373, -97.904, 49.277, 107.534, 25, -90]
  Set speed (16.7 mm/s)
  MoveL 2151 to (-74.99, 0.23, 131.08) mm, rotated rx 149.51 ry 0 rz 90.67 deg; joints [138.657, -9.285, 18.362, -97.902, 49.285, 107.505, 25, -90.672]
  MoveL 2152 to (-75.02, -0.11, 131.07) mm, rotated rx 149.73 ry 0 rz 92.05 deg; joints [138.741, -9.256, 18.329, -97.876, 49.367, 107.265, 25, -92.048]
  MoveL 2153 to (-73.47, -2, 131.92) mm, rotated rx 149.99 ry 0 rz 92.04 deg; joints [138.786, -9.051, 18.137, -97.875, 49.413, 107.007, 25, -92.041]
  MoveL 2154 to (-72.96, -2.95, 132.2) mm, rotated rx 149.99 ry 0 rz 92.04 deg; joints [138.774, -9.003, 18.093, -97.882, 49.401, 107.015, 25, -92.041]
  MoveL 2155 to (-72.33, -5.36, 132.45) mm, rotated rx 150.41 ry 0 rz 94.71 deg; joints [138.897, -8.876, 17.969, -97.85, 49.522, 106.585, 25, -94.709]
  MoveL 2156 to (-71.43, -6.39, 132.9) mm, rotated rx 150.78 ry 0 rz 95.6 deg; joints [138.996, -8.722, 17.822, -97.829, 49.62, 106.207, 25, -95.601]
  MoveL 2157 to (-70.8, -7.68, 133.18) mm, rotated rx 150.78 ry 0 rz 95.6 deg; joints [138.974, -8.663, 17.768, -97.84, 49.6, 106.219, 25, -95.601]
  MoveL 2158 to (-70.31, -9.65, 133.31) mm, rotated rx 150.89 ry 0 rz 97.24 deg; joints [139.006, -8.614, 17.722, -97.833, 49.63, 106.098, 25, -97.236]
  MoveL 2159 to (-70.2, -10.42, 133.32) mm, rotated rx 150.9 ry 0 rz 97.39 deg; joints [138.993, -8.594, 17.704, -97.839, 49.618, 106.096, 25, -97.392]
  MoveL 2160 to (-70.14, -12.43, 133.18) mm, rotated rx 150.79 ry 0 rz 99.04 deg; joints [138.965, -8.641, 17.748, -97.844, 49.591, 106.204, 25, -99.037]
  MoveL 2161 to (-69.55, -15.84, 133.12) mm, rotated rx 150.75 ry 0 rz 102.05 deg; joints [138.961, -8.667, 17.772, -97.844, 49.587, 106.242, 25, -102.049]
  MoveL 2162 to (-69.76, -17.49, 132.81) mm, rotated rx 150.75 ry 0 rz 102.05 deg; joints [138.908, -8.641, 17.751, -97.862, 49.536, 106.257, 25, -102.049]
  MoveL 2163 to (-70.51, -19.37, 132.15) mm, rotated rx 150.01 ry 0 rz 104.28 deg; joints [138.748, -8.972, 18.066, -97.892, 49.377, 107.012, 25, -104.277]
  MoveL 2164 to (-70.5, -20.09, 132.05) mm, rotated rx 149.98 ry 0 rz 104.48 deg; joints [138.728, -8.973, 18.068, -97.898, 49.357, 107.041, 25, -104.483]
  MoveL 2165 to (-70.76, -22.23, 131.56) mm, rotated rx 149.53 ry 0 rz 106.88 deg; joints [138.635, -9.192, 18.276, -97.915, 49.265, 107.502, 25, -106.881]
  MoveL 2166 to (-70.5, -23, 131.56) mm, rotated rx 149.53 ry 0 rz 107.51 deg; joints [138.637, -9.19, 18.274, -97.914, 49.267, 107.495, 25, -107.508]
  MoveL 2167 to (-70.37, -23.62, 131.53) mm, rotated rx 149.53 ry 0 rz 107.51 deg; joints [138.62, -9.173, 18.26, -97.921, 49.25, 107.501, 25, -107.508]
  MoveL 2168 to (-70.33, -24.58, 131.38) mm, rotated rx 149.5 ry 0 rz 107.8 deg; joints [138.592, -9.179, 18.267, -97.93, 49.223, 107.544, 25, -107.805]
  MoveL 2169 to (-70.61, -28.42, 130.45) mm, rotated rx 148.78 ry 0 rz 110.56 deg; joints [138.401, -9.479, 18.559, -97.976, 49.035, 108.279, 25, -110.56]
  MoveL 2170 to (-70.7, -29.36, 130.19) mm, rotated rx 148.72 ry 0 rz 110.83 deg; joints [138.363, -9.502, 18.584, -97.988, 48.999, 108.353, 25, -110.827]
  MoveL 2171 to (-71.43, -32.36, 129.07) mm, rotated rx 147.88 ry 0 rz 112.73 deg; joints [138.134, -9.854, 18.931, -98.047, 48.774, 109.231, 25, -112.734]
  Set speed (16.7 mm/s)
  MoveL 2172 to (-81.24, -36.47, 146.01) mm, rotated rx 147.88 ry 0 rz 112.73 deg; joints [138.079, -9.962, 18.316, -97.432, 48.622, 108.286, 25, -112.734]
  Set speed (1000.0 mm/s)
  MoveL 2173 to (-77.22, -38.49, 147.66) mm, rotated rx 148.8 ry 0 rz 115.82 deg; joints [138.379, -9.591, 17.945, -97.356, 48.917, 107.319, 25, -115.822]
  Set speed (5.0 mm/s)
  MoveL 2174 to (-67.89, -33.98, 130.56) mm, rotated rx 148.8 ry 0 rz 115.82 deg; joints [138.427, -9.493, 18.57, -97.966, 49.061, 108.26, 25, -115.822]
  Set speed (16.7 mm/s)
  MoveL 2175 to (-67.23, -36.01, 130.36) mm, rotated rx 148.65 ry 0 rz 117.44 deg; joints [138.387, -9.556, 18.632, -97.976, 49.021, 108.416, 25, -117.439]
  MoveL 2176 to (-67.2, -37.94, 129.81) mm, rotated rx 148.3 ry 0 rz 119.8 deg; joints [138.326, -9.75, 18.817, -97.986, 48.96, 108.761, 25, -119.803]
  MoveL 2177 to (-66.35, -38.67, 130.04) mm, rotated rx 148.47 ry 0 rz 120.6 deg; joints [138.374, -9.678, 18.747, -97.974, 49.007, 108.58, 25, -120.604]
  MoveL 2178 to (-65.37, -39.02, 130.42) mm, rotated rx 148.93 ry 0 rz 121.71 deg; joints [138.505, -9.523, 18.593, -97.938, 49.136, 108.103, 25, -121.708]
  MoveL 2179 to (-64.59, -39.53, 130.67) mm, rotated rx 148.93 ry 0 rz 121.71 deg; joints [138.494, -9.481, 18.555, -97.944, 49.126, 108.11, 25, -121.708]
  MoveL 2180 to (-64.18, -39.97, 130.74) mm, rotated rx 148.94 ry 0 rz 121.78 deg; joints [138.487, -9.458, 18.533, -97.948, 49.119, 108.102, 25, -121.78]
  MoveL 2181 to (-63.7, -40.59, 130.77) mm, rotated rx 148.97 ry 0 rz 122.38 deg; joints [138.496, -9.445, 18.521, -97.946, 49.128, 108.068, 25, -122.376]
  MoveL 2182 to (-62.85, -41.02, 131.05) mm, rotated rx 149.31 ry 0 rz 123.77 deg; joints [138.607, -9.344, 18.419, -97.915, 49.236, 107.708, 25, -123.77]
  MoveL 2183 to (-61.73, -42.25, 131.2) mm, rotated rx 149.31 ry 0 rz 123.77 deg; joints [138.572, -9.285, 18.367, -97.93, 49.203, 107.723, 25, -123.77]
  MoveL 2184 to (-61.42, -43.97, 130.78) mm, rotated rx 149.03 ry 0 rz 125.97 deg; joints [138.525, -9.445, 18.519, -97.936, 49.156, 108.002, 25, -125.965]
  MoveL 2185 to (-60.94, -44.4, 130.86) mm, rotated rx 149.05 ry 0 rz 126.05 deg; joints [138.519, -9.419, 18.495, -97.94, 49.15, 107.991, 25, -126.051]
  MoveL 2186 to (-60.17, -45.41, 130.87) mm, rotated rx 149.05 ry 0 rz 126.78 deg; joints [138.512, -9.408, 18.485, -97.943, 49.144, 107.991, 25, -126.777]
  MoveL 2187 to (-58.97, -46.12, 131.16) mm, rotated rx 149.35 ry 0 rz 128.53 deg; joints [138.615, -9.319, 18.396, -97.914, 49.244, 107.672, 25, -128.53]
  MoveL 2188 to (-57.34, -45.99, 131.92) mm, rotated rx 149.74 ry 0 rz 129.2 deg; joints [138.73, -9.136, 18.219, -97.887, 49.358, 107.271, 25, -129.202]
  MoveL 2189 to (-55.9, -47.06, 132.17) mm, rotated rx 150.12 ry 0 rz 129.89 deg; joints [138.802, -8.966, 18.057, -97.875, 49.429, 106.885, 25, -129.89]
  MoveL 2190 to (-53.58, -50.2, 131.97) mm, rotated rx 149.97 ry 0 rz 132.92 deg; joints [138.76, -9.031, 18.119, -97.884, 49.388, 107.043, 25, -132.924]
  MoveL 2191 to (-52.99, -49.57, 132.45) mm, rotated rx 151.13 ry 0 rz 135.03 deg; joints [139.097, -8.69, 17.787, -97.8, 49.718, 105.829, 25, -135.029]
  MoveL 2192 to (-52.53, -49.31, 132.73) mm, rotated rx 151.19 ry 0 rz 135.05 deg; joints [139.12, -8.646, 17.746, -97.795, 49.741, 105.768, 25, -135.049]
  MoveL 2193 to (-49.78, -48.12, 134.21) mm, rotated rx 152.41 ry 0 rz 135.97 deg; joints [139.442, -8.131, 17.261, -97.734, 50.061, 104.535, 25, -135.968]
  MoveL 2194 to (-48.98, -47.93, 134.58) mm, rotated rx 152.41 ry 0 rz 135.97 deg; joints [139.448, -8.09, 17.224, -97.735, 50.067, 104.538, 25, -135.968]
  MoveL 2195 to (-47.83, -48.01, 134.96) mm, rotated rx 152.53 ry 0 rz 136.19 deg; joints [139.475, -8.003, 17.144, -97.733, 50.094, 104.423, 25, -136.187]
  MoveL 2196 to (-46.35, -49.06, 135.1) mm, rotated rx 152.53 ry 0 rz 136.19 deg; joints [139.437, -7.94, 17.087, -97.749, 50.058, 104.438, 25, -136.187]
  MoveL 2197 to (-44.24, -51.83, 134.77) mm, rotated rx 152.25 ry 0 rz 139.09 deg; joints [139.364, -8.058, 17.197, -97.762, 49.985, 104.718, 25, -139.095]
  Set speed (16.7 mm/s)
  MoveL 2198 to (-50.34, -58.87, 152.47) mm, rotated rx 152.25 ry 0 rz 139.09 deg; joints [139.343, -8.117, 16.536, -97.167, 49.872, 103.789, 25, -139.095]
  Set speed (1000.0 mm/s)
  MoveL 2199 to (-44.65, -61.37, 153.25) mm, rotated rx 153.05 ry 0 rz 145.25 deg; joints [139.602, -7.854, 16.289, -97.116, 50.127, 102.97, 25, -145.25]
  Set speed (5.0 mm/s)
  MoveL 2200 to (-39.49, -53.93, 135.43) mm, rotated rx 153.05 ry 0 rz 145.25 deg; joints [139.616, -7.805, 16.959, -97.707, 50.234, 103.896, 25, -145.25]
  Set speed (16.7 mm/s)
  MoveL 2201 to (-37.74, -54.13, 135.84) mm, rotated rx 153.16 ry 0 rz 145.51 deg; joints [139.627, -7.699, 16.863, -97.711, 50.245, 103.798, 25, -145.505]
  MoveL 2202 to (-36.32, -54.77, 135.96) mm, rotated rx 153.27 ry 0 rz 146.84 deg; joints [139.655, -7.652, 16.82, -97.707, 50.274, 103.688, 25, -146.839]
  Set speed (16.7 mm/s)
  MoveL 2203 to (-41.25, -62.3, 153.82) mm, rotated rx 153.27 ry 0 rz 146.84 deg; joints [139.643, -7.699, 16.148, -97.117, 50.169, 102.762, 25, -146.839]
  Set speed (1000.0 mm/s)
  MoveL 2204 to (-38.06, -61.38, 155.02) mm, rotated rx 154.24 ry 0 rz 148.89 deg; joints [139.911, -7.289, 15.772, -97.078, 50.437, 101.792, 25, -148.886]
  Set speed (5.0 mm/s)
  MoveL 2205 to (-33.57, -53.93, 137.01) mm, rotated rx 154.24 ry 0 rz 148.89 deg; joints [139.917, -7.253, 16.454, -97.664, 50.534, 102.714, 25, -148.886]
  Set speed (16.7 mm/s)
  MoveL 2206 to (-29.71, -54.62, 137.63) mm, rotated rx 154.81 ry 0 rz 152.27 deg; joints [140.063, -7.011, 16.234, -97.643, 50.68, 102.153, 25, -152.274]
  MoveL 2207 to (-27.31, -54.41, 138.2) mm, rotated rx 155.44 ry 0 rz 154.32 deg; joints [140.225, -6.749, 15.999, -97.621, 50.843, 101.52, 25, -154.32]
  MoveL 2208 to (-25.95, -54.63, 138.38) mm, rotated rx 155.44 ry 0 rz 154.32 deg; joints [140.201, -6.696, 15.951, -97.632, 50.82, 101.531, 25, -154.32]
  MoveL 2209 to (-24.86, -55.33, 138.3) mm, rotated rx 155.45 ry 0 rz 154.54 deg; joints [140.172, -6.67, 15.928, -97.642, 50.792, 101.535, 25, -154.544]
  MoveL 2210 to (-24.2, -56.01, 138.15) mm, rotated rx 155.3 ry 0 rz 155.4 deg; joints [140.135, -6.735, 15.986, -97.646, 50.755, 101.681, 25, -155.399]
  MoveL 2211 to (-24.17, -55.99, 138.16) mm, rotated rx 155.58 ry 0 rz 158.39 deg; joints [140.27, -6.731, 15.983, -97.611, 50.887, 101.382, 25, -158.388]
  MoveL 2212 to (-23.49, -55.66, 138.41) mm, rotated rx 155.82 ry 0 rz 158.9 deg; joints [140.332, -6.628, 15.892, -97.603, 50.949, 101.146, 25, -158.904]
  MoveL 2213 to (-22.23, -55.42, 138.72) mm, rotated rx 155.82 ry 0 rz 158.9 deg; joints [140.321, -6.571, 15.84, -97.611, 50.939, 101.155, 25, -158.904]
  MoveL 2214 to (-21.13, -55.63, 138.8) mm, rotated rx 155.84 ry 0 rz 159.09 deg; joints [140.308, -6.529, 15.802, -97.618, 50.927, 101.136, 25, -159.094]
  MoveL 2215 to (-19.51, -56.29, 138.77) mm, rotated rx 155.82 ry 0 rz 160.78 deg; joints [140.302, -6.539, 15.811, -97.619, 50.921, 101.159, 25, -160.777]
  MoveL 2216 to (-18.07, -56.32, 138.96) mm, rotated rx 156.03 ry 0 rz 162.8 deg; joints [140.371, -6.472, 15.752, -97.606, 50.989, 100.948, 25, -162.803]
  MoveL 2217 to (-16.43, -56.97, 138.89) mm, rotated rx 156.03 ry 0 rz 162.8 deg; joints [140.325, -6.427, 15.711, -97.622, 50.944, 100.961, 25, -162.803]
  MoveL 2218 to (-15.77, -57.73, 138.66) mm, rotated rx 156 ry 0 rz 162.95 deg; joints [140.289, -6.436, 15.719, -97.63, 50.91, 100.993, 25, -162.947]
  MoveL 2219 to (-15.43, -58.46, 138.39) mm, rotated rx 155.45 ry 0 rz 165.1 deg; joints [140.207, -6.698, 15.953, -97.63, 50.826, 101.523, 25, -165.105]
  MoveL 2220 to (-12.07, -59.39, 138.33) mm, rotated rx 155.39 ry 0 rz 168.37 deg; joints [140.191, -6.722, 15.975, -97.632, 50.81, 101.582, 25, -168.365]
  MoveL 2221 to (-10.92, -60, 138.16) mm, rotated rx 155.39 ry 0 rz 168.37 deg; joints [140.152, -6.7, 15.954, -97.645, 50.771, 101.591, 25, -168.365]
  MoveL 2222 to (-10.46, -60.5, 137.98) mm, rotated rx 155.37 ry 0 rz 168.43 deg; joints [140.127, -6.708, 15.961, -97.65, 50.747, 101.613, 25, -168.435]
  MoveL 2223 to (-9.89, -61.32, 137.66) mm, rotated rx 155.07 ry 0 rz 169.13 deg; joints [140.051, -6.838, 16.079, -97.66, 50.671, 101.91, 25, -169.133]
  MoveL 2224 to (-9.41, -61.94, 137.41) mm, rotated rx 155 ry 0 rz 169.4 deg; joints [140.018, -6.872, 16.109, -97.666, 50.638, 101.978, 25, -169.396]
  MoveL 2225 to (-8.41, -64.13, 136.47) mm, rotated rx 154.15 ry 0 rz 170.65 deg; joints [139.797, -7.24, 16.443, -97.698, 50.418, 102.831, 25, -170.65]
  MoveL 2226 to (-7.46, -65.27, 135.98) mm, rotated rx 153.57 ry 0 rz 171.9 deg; joints [139.662, -7.484, 16.667, -97.718, 50.283, 103.408, 25, -171.901]
  MoveL 2227 to (-7.37, -65.37, 135.94) mm, rotated rx 153.23 ry 0 rz 173.81 deg; joints [139.643, -7.662, 16.828, -97.71, 50.262, 103.724, 25, -173.813]
  MoveL 2228 to (-6.73, -65.37, 135.97) mm, rotated rx 153.26 ry 0 rz 174.37 deg; joints [139.65, -7.649, 16.817, -97.708, 50.269, 103.695, 25, -174.37]
  MoveL 2229 to (-6.15, -65.42, 135.98) mm, rotated rx 153.26 ry 0 rz 174.62 deg; joints [139.643, -7.64, 16.809, -97.711, 50.262, 103.698, 25, -174.618]
  MoveL 2230 to (-3.34, -65.88, 135.85) mm, rotated rx 153.16 ry 0 rz 176.87 deg; joints [139.609, -7.679, 16.844, -97.718, 50.229, 103.806, 25, -176.874]
  MoveL 2231 to (-2.74, -66.04, 135.79) mm, rotated rx 153.16 ry 0 rz 176.87 deg; joints [139.591, -7.666, 16.833, -97.724, 50.211, 103.811, 25, -176.874]
  MoveL 2232 to (-1.69, -66.7, 135.48) mm, rotated rx 152.83 ry 0 rz 178.6 deg; joints [139.532, -7.825, 16.98, -97.729, 50.152, 104.127, 25, -178.596]
  MoveL 2233 to (-0.75, -66.76, 135.46) mm, rotated rx 152.84 ry 0 rz 178.91 deg; joints [139.518, -7.809, 16.965, -97.735, 50.138, 104.129, 25, -178.911]
  MoveL 2234 to (-0.36, -66.92, 135.38) mm, rotated rx 152.95 ry 0 rz -179 deg; joints [139.589, -7.835, 16.988, -97.712, 50.208, 103.995, 25, -180.999]
  MoveL 2235 to (0.64, -66.19, 135.74) mm, rotated rx 153.26 ry 0 rz -178.12 deg; joints [139.671, -7.704, 16.866, -97.699, 50.289, 103.684, 25, -181.883]
  MoveL 2236 to (1.78, -65.71, 135.97) mm, rotated rx 153.26 ry 0 rz -178.12 deg; joints [139.652, -7.652, 16.82, -97.708, 50.271, 103.694, 25, -181.883]
  MoveL 2237 to (2.93, -65.71, 135.95) mm, rotated rx 153.27 ry 0 rz -178.02 deg; joints [139.627, -7.621, 16.792, -97.717, 50.247, 103.696, 25, -181.979]
  MoveL 2238 to (4, -65.92, 135.82) mm, rotated rx 153.16 ry 0 rz -177.1 deg; joints [139.598, -7.669, 16.836, -97.722, 50.218, 103.809, 25, -182.899]
  MoveL 2239 to (7.3, -65.68, 135.79) mm, rotated rx 153.09 ry 0 rz -173.46 deg; joints [139.604, -7.72, 16.882, -97.716, 50.224, 103.87, 25, -186.536]
  MoveL 2240 to (8.4, -65.81, 135.67) mm, rotated rx 153.09 ry 0 rz -173.46 deg; joints [139.572, -7.698, 16.863, -97.727, 50.192, 103.879, 25, -186.536]
  MoveL 2241 to (9.29, -66.23, 135.4) mm, rotated rx 153.05 ry 0 rz -173.3 deg; joints [139.535, -7.712, 16.876, -97.737, 50.156, 103.923, 25, -186.698]
  MoveL 2242 to (11.54, -67.79, 134.45) mm, rotated rx 152.22 ry 0 rz -171.54 deg; joints [139.319, -8.066, 17.206, -97.775, 49.941, 104.762, 25, -188.458]
  MoveL 2243 to (12, -68.18, 134.21) mm, rotated rx 152.14 ry 0 rz -171.42 deg; joints [139.285, -8.102, 17.24, -97.783, 49.908, 104.843, 25, -188.575]
  MoveL 2244 to (12.74, -68.99, 133.73) mm, rotated rx 151.8 ry 0 rz -171.01 deg; joints [139.19, -8.247, 17.376, -97.801, 49.813, 105.184, 25, -188.989]
  MoveL 2245 to (13.57, -68.32, 134) mm, rotated rx 151.56 ry 0 rz -167.97 deg; joints [139.219, -8.393, 17.509, -97.782, 49.841, 105.409, 25, -192.027]
  MoveL 2246 to (14.06, -68.11, 134.06) mm, rotated rx 151.6 ry 0 rz -167.53 deg; joints [139.232, -8.373, 17.49, -97.78, 49.853, 105.36, 25, -192.47]
  MoveL 2247 to (18.3, -67.01, 134.08) mm, rotated rx 151.6 ry 0 rz -164.33 deg; joints [139.221, -8.357, 17.476, -97.785, 49.842, 105.37, 25, -195.673]
  MoveL 2248 to (18.46, -66.21, 134.47) mm, rotated rx 151.82 ry 0 rz -163.74 deg; joints [139.292, -8.266, 17.39, -97.769, 49.913, 105.146, 25, -196.261]
  MoveL 2249 to (19.9, -64.86, 134.93) mm, rotated rx 152.3 ry 0 rz -162.37 deg; joints [139.411, -8.065, 17.202, -97.748, 50.031, 104.658, 25, -197.628]
  MoveL 2250 to (20.58, -64.61, 134.95) mm, rotated rx 152.32 ry 0 rz -161.75 deg; joints [139.415, -8.059, 17.196, -97.747, 50.035, 104.642, 25, -198.25]
  MoveL 2251 to (26.87, -62.57, 134.8) mm, rotated rx 152.17 ry 0 rz -156.31 deg; joints [139.374, -8.114, 17.248, -97.755, 49.995, 104.79, 25, -203.69]
  MoveL 2252 to (28.7, -61.62, 134.86) mm, rotated rx 152.22 ry 0 rz -154.32 deg; joints [139.394, -8.103, 17.237, -97.75, 50.014, 104.741, 25, -205.681]
  MoveL 2253 to (29.82, -61.29, 134.76) mm, rotated rx 152.22 ry 0 rz -154.32 deg; joints [139.361, -8.076, 17.214, -97.762, 49.982, 104.752, 25, -205.681]
  MoveL 2254 to (30.96, -61.36, 134.47) mm, rotated rx 152.17 ry 0 rz -154.12 deg; joints [139.32, -8.089, 17.227, -97.773, 49.942, 104.8, 25, -205.879]
  MoveL 2255 to (32.73, -61.9, 133.81) mm, rotated rx 151.32 ry 0 rz -151.85 deg; joints [139.146, -8.466, 17.579, -97.8, 49.769, 105.649, 25, -208.152]
  MoveL 2256 to (34.2, -61.35, 133.7) mm, rotated rx 151.22 ry 0 rz -150.55 deg; joints [139.12, -8.509, 17.62, -97.805, 49.743, 105.752, 25, -209.452]
  MoveL 2257 to (34.89, -61.18, 133.6) mm, rotated rx 151.2 ry 0 rz -150.41 deg; joints [139.097, -8.51, 17.621, -97.812, 49.721, 105.783, 25, -209.586]
  MoveL 2258 to (35.94, -61.16, 133.33) mm, rotated rx 150.91 ry 0 rz -148.66 deg; joints [139.055, -8.664, 17.765, -97.814, 49.678, 106.069, 25, -211.342]
  MoveL 2259 to (37.28, -60.11, 133.44) mm, rotated rx 150.99 ry 0 rz -147.26 deg; joints [139.079, -8.628, 17.731, -97.809, 49.701, 105.982, 25, -212.737]
  MoveL 2260 to (37.77, -59.72, 133.48) mm, rotated rx 151.02 ry 0 rz -146.77 deg; joints [139.085, -8.616, 17.72, -97.808, 49.708, 105.955, 25, -213.226]
  MoveL 2261 to (38.36, -59.36, 133.47) mm, rotated rx 151.02 ry 0 rz -146.77 deg; joints [139.068, -8.596, 17.702, -97.815, 49.691, 105.962, 25, -213.226]
  MoveL 2262 to (43.48, -56.74, 133.04) mm, rotated rx 150.64 ry 0 rz -142.12 deg; joints [138.97, -8.756, 17.854, -97.835, 49.594, 106.347, 25, -217.878]
  MoveL 2263 to (44.61, -56.39, 132.8) mm, rotated rx 150.64 ry 0 rz -142.12 deg; joints [138.932, -8.739, 17.841, -97.848, 49.558, 106.358, 25, -217.878]
  MoveL 2264 to (45.13, -56.35, 132.64) mm, rotated rx 150.55 ry 0 rz -141.89 deg; joints [138.903, -8.775, 17.876, -97.855, 49.529, 106.449, 25, -218.111]
  MoveL 2265 to (47.13, -56.37, 131.95) mm, rotated rx 149.73 ry 0 rz -139.33 deg; joints [138.74, -9.148, 18.229, -97.883, 49.367, 107.271, 25, -220.666]
  MoveL 2266 to (50.68, -53.13, 131.95) mm, rotated rx 150.39 ry 0 rz -136.58 deg; joints [138.849, -8.89, 17.985, -97.865, 49.475, 106.611, 25, -223.419]
  MoveL 2267 to (51.14, -52.77, 131.92) mm, rotated rx 150.38 ry 0 rz -136.49 deg; joints [138.834, -8.881, 17.977, -97.87, 49.461, 106.624, 25, -223.513]
  MoveL 2268 to (52.56, -50.63, 132.2) mm, rotated rx 150.61 ry 0 rz -134.48 deg; joints [138.897, -8.787, 17.887, -97.856, 49.523, 106.39, 25, -225.519]
  Set speed (16.7 mm/s)
  MoveL 2269 to (59.81, -57.33, 149.59) mm, rotated rx 150.59 ry 0 rz -134.26 deg; joints [138.858, -8.874, 17.251, -97.254, 49.39, 105.474, 25, -225.736]
  Set speed (1000.0 mm/s)
  MoveL 2270 to (61.99, -54.39, 149.8) mm, rotated rx 150.73 ry 0 rz -131.5 deg; joints [138.906, -8.823, 17.202, -97.243, 49.437, 105.329, 25, -228.501]
  Set speed (5.0 mm/s)
  MoveL 2271 to (54.66, -47.91, 132.36) mm, rotated rx 150.73 ry 0 rz -131.5 deg; joints [138.938, -8.747, 17.848, -97.846, 49.563, 106.264, 25, -228.501]
  Set speed (16.7 mm/s)
  MoveL 2272 to (55.79, -46.79, 132.29) mm, rotated rx 150.67 ry 0 rz -130.2 deg; joints [138.925, -8.772, 17.872, -97.848, 49.55, 106.321, 25, -229.797]
  MoveL 2273 to (56.07, -46.15, 132.39) mm, rotated rx 150.78 ry 0 rz -129.06 deg; joints [138.971, -8.754, 17.853, -97.835, 49.595, 106.208, 25, -230.945]
  MoveL 2274 to (56.83, -45.24, 132.38) mm, rotated rx 150.78 ry 0 rz -129.06 deg; joints [138.941, -8.719, 17.822, -97.847, 49.566, 106.219, 25, -230.945]
  MoveL 2275 to (57.77, -44.66, 132.18) mm, rotated rx 150.75 ry 0 rz -128.83 deg; joints [138.907, -8.721, 17.825, -97.858, 49.533, 106.256, 25, -231.172]
  MoveL 2276 to (60.3, -43.63, 131.38) mm, rotated rx 150.12 ry 0 rz -126.92 deg; joints [138.74, -8.988, 18.081, -97.894, 49.369, 106.901, 25, -233.085]
  MoveL 2277 to (61.86, -41.57, 131.32) mm, rotated rx 149.91 ry 0 rz -123.88 deg; joints [138.726, -9.103, 18.188, -97.891, 49.354, 107.104, 25, -236.117]
  MoveL 2278 to (62.57, -39.87, 131.52) mm, rotated rx 150.07 ry 0 rz -122 deg; joints [138.785, -9.055, 18.141, -97.875, 49.411, 106.933, 25, -237.997]
  MoveL 2279 to (63.23, -38.94, 131.48) mm, rotated rx 150.07 ry 0 rz -122 deg; joints [138.755, -9.023, 18.113, -97.887, 49.382, 106.944, 25, -237.997]
  MoveL 2280 to (63.85, -38.47, 131.32) mm, rotated rx 150.05 ry 0 rz -121.91 deg; joints [138.73, -9.021, 18.112, -97.895, 49.358, 106.965, 25, -238.09]
  MoveL 2281 to (64.49, -38.1, 131.11) mm, rotated rx 149.89 ry 0 rz -121.39 deg; joints [138.686, -9.09, 18.179, -97.905, 49.315, 107.134, 25, -238.611]
  MoveL 2282 to (64.68, -37.79, 131.11) mm, rotated rx 149.74 ry 0 rz -120.25 deg; joints [138.682, -9.174, 18.257, -97.901, 49.311, 107.276, 25, -239.753]
  MoveL 2283 to (65.32, -37.14, 130.98) mm, rotated rx 149.74 ry 0 rz -120.25 deg; joints [138.654, -9.156, 18.242, -97.911, 49.284, 107.285, 25, -239.753]
  MoveL 2284 to (65.81, -36.84, 130.82) mm, rotated rx 149.72 ry 0 rz -120.18 deg; joints [138.633, -9.161, 18.248, -97.918, 49.263, 107.308, 25, -239.822]
  MoveL 2285 to (66.52, -36.5, 130.55) mm, rotated rx 149.51 ry 0 rz -119.66 deg; joints [138.578, -9.248, 18.333, -97.931, 49.209, 107.523, 25, -240.335]
  MoveL 2286 to (70.08, -32.64, 129.71) mm, rotated rx 148.7 ry 0 rz -115.16 deg; joints [138.389, -9.603, 18.676, -97.973, 49.023, 108.359, 25, -244.839]
  MoveL 2287 to (70.59, -32.15, 129.55) mm, rotated rx 148.63 ry 0 rz -114.92 deg; joints [138.361, -9.624, 18.698, -97.981, 48.995, 108.429, 25, -245.08]
  MoveL 2288 to (72.16, -30.71, 129.03) mm, rotated rx 148.24 ry 0 rz -113.43 deg; joints [138.256, -9.788, 18.86, -98.008, 48.892, 108.837, 25, -246.569]
  MoveL 2289 to (72.5, -29.55, 129.13) mm, rotated rx 148.2 ry 0 rz -111.83 deg; joints [138.275, -9.827, 18.894, -97.999, 48.91, 108.87, 25, -248.171]
  MoveL 2290 to (72.86, -28.78, 129.09) mm, rotated rx 148.17 ry 0 rz -111.19 deg; joints [138.268, -9.839, 18.905, -98.001, 48.903, 108.898, 25, -248.808]
  MoveL 2291 to (73.21, -28.21, 129.02) mm, rotated rx 148.17 ry 0 rz -111.19 deg; joints [138.248, -9.823, 18.892, -98.009, 48.885, 108.905, 25, -248.808]
  MoveL 2292 to (79.18, -19.42, 127.09) mm, rotated rx 146.78 ry 0 rz -103.76 deg; joints [137.869, -10.406, 19.474, -98.113, 48.513, 110.367, 25, -256.241]
  MoveL 2293 to (84.02, -9.55, 125.11) mm, rotated rx 145.33 ry 0 rz -96.25 deg; joints [137.476, -11.005, 20.08, -98.231, 48.13, 111.896, 25, -263.746]
  MoveL 2294 to (85.47, -8.13, 124.22) mm, rotated rx 145.33 ry 0 rz -96.25 deg; joints [137.401, -11.008, 20.092, -98.26, 48.058, 111.922, 25, -263.746]
  MoveL 2295 to (86.56, -8.17, 123.47) mm, rotated rx 145.33 ry 0 rz -96.25 deg; joints [137.369, -11.049, 20.135, -98.271, 48.027, 111.931, 25, -263.746]
  MoveL 2296 to (87.6, -9.12, 122.67) mm, rotated rx 145.33 ry 0 rz -96.25 deg; joints [137.358, -11.121, 20.204, -98.271, 48.016, 111.929, 25, -263.746]
  MoveL 2297 to (87.88, -11, 122.34) mm, rotated rx 145.33 ry 0 rz -96.25 deg; joints [137.391, -11.197, 20.272, -98.255, 48.047, 111.912, 25, -263.746]
  MoveL 2298 to (85.96, -19.02, 122.71) mm, rotated rx 145.61 ry 0 rz -101.73 deg; joints [137.461, -11.081, 20.153, -98.233, 48.116, 111.621, 25, -258.271]
  MoveL 2299 to (82.72, -28.28, 123.17) mm, rotated rx 145.94 ry 0 rz -108.29 deg; joints [137.545, -10.942, 20.012, -98.207, 48.197, 111.273, 25, -251.707]
  MoveL 2300 to (79.9, -32.89, 123.88) mm, rotated rx 146.4 ry 0 rz -111.61 deg; joints [137.683, -10.757, 19.822, -98.163, 48.332, 110.772, 25, -248.392]
  MoveL 2301 to (79.79, -32.88, 123.91) mm, rotated rx 144.76 ry 0 rz -113.13 deg; joints [137.265, -11.213, 20.303, -98.305, 47.926, 112.528, 25, -246.868]
  MoveL 2302 to (81.28, -31.88, 123.21) mm, rotated rx 144.28 ry 0 rz -112.11 deg; joints [137.13, -11.41, 20.507, -98.35, 47.796, 113.046, 25, -247.894]
  MoveL 2303 to (83.27, -31.68, 121.93) mm, rotated rx 144.25 ry 0 rz -112.16 deg; joints [137.049, -11.458, 20.564, -98.381, 47.717, 113.1, 25, -247.838]
  MoveL 2304 to (84.18, -32.65, 121.06) mm, rotated rx 144.23 ry 0 rz -112.2 deg; joints [137.023, -11.528, 20.634, -98.388, 47.693, 113.122, 25, -247.801]
  MoveL 2305 to (84.06, -35.02, 120.5) mm, rotated rx 144.21 ry 0 rz -112.26 deg; joints [137.049, -11.636, 20.732, -98.373, 47.716, 113.133, 25, -247.742]
  MoveL 2306 to (83.49, -36.19, 120.53) mm, rotated rx 144.05 ry 0 rz -114.11 deg; joints [136.973, -11.633, 20.741, -98.405, 47.644, 113.323, 25, -245.891]
  MoveL 2307 to (83.76, -38.69, 119.57) mm, rotated rx 143.44 ry 0 rz -115.48 deg; joints [136.799, -11.876, 20.998, -98.468, 47.476, 113.982, 25, -244.516]
  MoveL 2308 to (85.01, -41.41, 117.75) mm, rotated rx 142.04 ry 0 rz -117 deg; joints [136.4, -12.394, 21.556, -98.622, 47.092, 115.517, 25, -242.998]
  MoveL 2309 to (84.94, -43.5, 117.06) mm, rotated rx 142.04 ry 0 rz -117 deg; joints [136.421, -12.49, 21.645, -98.609, 47.112, 115.502, 25, -242.998]
  MoveL 2310 to (84.41, -44.47, 117.08) mm, rotated rx 142.03 ry 0 rz -117.2 deg; joints [136.439, -12.517, 21.667, -98.6, 47.129, 115.502, 25, -242.803]
  MoveL 2311 to (82.72, -46.56, 117.46) mm, rotated rx 142.26 ry 0 rz -118.78 deg; joints [136.507, -12.424, 21.568, -98.574, 47.193, 115.247, 25, -241.215]
  MoveL 2312 to (82.46, -48.44, 116.89) mm, rotated rx 141.93 ry 0 rz -120.43 deg; joints [136.385, -12.528, 21.687, -98.624, 47.077, 115.627, 25, -239.57]
  MoveL 2313 to (82.16, -49.29, 116.74) mm, rotated rx 141.81 ry 0 rz -121.21 deg; joints [136.343, -12.558, 21.724, -98.642, 47.037, 115.76, 25, -238.792]
  MoveL 2314 to (82.94, -48.44, 116.52) mm, rotated rx 139.92 ry 0 rz -120.85 deg; joints [135.889, -13.139, 22.366, -98.835, 46.603, 117.826, 25, -239.146]
  MoveL 2315 to (83.88, -47.94, 116.06) mm, rotated rx 139.87 ry 0 rz -120.71 deg; joints [135.843, -13.156, 22.391, -98.857, 46.559, 117.899, 25, -239.287]
  MoveL 2316 to (86.1, -47.26, 114.71) mm, rotated rx 139.06 ry 0 rz -119.72 deg; joints [135.606, -13.471, 22.743, -98.965, 46.334, 118.81, 25, -240.279]
  MoveL 2317 to (87.26, -46.57, 114.11) mm, rotated rx 138.59 ry 0 rz -118.87 deg; joints [135.484, -13.652, 22.944, -99.021, 46.218, 119.33, 25, -241.133]
  MoveL 2318 to (88.1, -46.23, 113.6) mm, rotated rx 138.26 ry 0 rz -118.78 deg; joints [135.373, -13.761, 23.074, -99.075, 46.114, 119.719, 25, -241.216]
  MoveL 2319 to (89.65, -47.03, 112.04) mm, rotated rx 137.49 ry 0 rz -118.6 deg; joints [135.146, -14.075, 23.43, -99.187, 45.9, 120.592, 25, -241.403]
  MoveL 2320 to (90.94, -46.5, 111.23) mm, rotated rx 137.02 ry 0 rz -117.97 deg; joints [135.008, -14.256, 23.638, -99.257, 45.769, 121.133, 25, -242.028]
  MoveL 2321 to (92.41, -46.56, 109.99) mm, rotated rx 137.02 ry 0 rz -117.97 deg; joints [134.948, -14.291, 23.687, -99.288, 45.713, 121.164, 25, -242.028]
  Set speed (16.7 mm/s)
  MoveL 2322 to (104.65, -53.08, 124.41) mm, rotated rx 136.91 ry 0 rz -117.98 deg; joints [134.76, -14.563, 23.24, -98.65, 45.418, 120.314, 25, -242.019]
  Set speed (1000.0 mm/s)
  MoveL 2323 to (106.64, -54.76, 121.97) mm, rotated rx 135.66 ry 0 rz -118.25 deg; joints [134.379, -15.044, 23.803, -98.845, 45.058, 121.762, 25, -241.748]
  Set speed (5.0 mm/s)
  MoveL 2324 to (94.32, -48.14, 107.66) mm, rotated rx 135.66 ry 0 rz -118.25 deg; joints [134.549, -14.797, 24.281, -99.503, 45.339, 122.733, 25, -241.748]
  Set speed (16.7 mm/s)
  MoveL 2325 to (94.76, -48.45, 107.15) mm, rotated rx 135.6 ry 0 rz -118.25 deg; joints [134.517, -14.841, 24.333, -99.52, 45.309, 122.818, 25, -241.748]
  MoveL 2326 to (95.38, -49.1, 106.29) mm, rotated rx 135.13 ry 0 rz -118.4 deg; joints [134.379, -15.014, 24.539, -99.599, 45.18, 123.361, 25, -241.597]
  MoveL 2327 to (96.58, -49.18, 105.16) mm, rotated rx 134.03 ry 0 rz -118.12 deg; joints [134.081, -15.384, 24.986, -99.772, 44.904, 124.638, 25, -241.879]
  MoveL 2328 to (97.3, -49.5, 104.35) mm, rotated rx 134.03 ry 0 rz -118.12 deg; joints [134.052, -15.416, 25.025, -99.79, 44.877, 124.656, 25, -241.879]
  MoveL 2329 to (97.87, -50.47, 103.35) mm, rotated rx 133.95 ry 0 rz -118.14 deg; joints [134.014, -15.499, 25.118, -99.813, 44.841, 124.759, 25, -241.859]
  MoveL 2330 to (98.14, -51.93, 102.37) mm, rotated rx 133.43 ry 0 rz -118.75 deg; joints [133.858, -15.687, 25.35, -99.908, 44.697, 125.373, 25, -241.254]
  MoveL 2331 to (97.89, -53.62, 101.74) mm, rotated rx 133.43 ry 0 rz -118.75 deg; joints [133.877, -15.767, 25.424, -99.895, 44.715, 125.36, 25, -241.254]
  MoveL 2332 to (96.76, -55.02, 102.08) mm, rotated rx 133.43 ry 0 rz -118.75 deg; joints [133.933, -15.814, 25.454, -99.86, 44.767, 125.324, 25, -241.254]
  MoveL 2333 to (96.07, -55.49, 102.48) mm, rotated rx 133.64 ry 0 rz -119.14 deg; joints [133.996, -15.736, 25.359, -99.822, 44.825, 125.073, 25, -240.865]
  MoveL 2334 to (88.95, -59.16, 106.76) mm, rotated rx 135.86 ry 0 rz -122.64 deg; joints [134.667, -14.913, 24.366, -99.434, 45.449, 122.464, 25, -237.361]
  MoveL 2335 to (88.14, -59.55, 107.21) mm, rotated rx 136.12 ry 0 rz -123.06 deg; joints [134.744, -14.816, 24.251, -99.392, 45.521, 122.161, 25, -236.939]
  MoveL 2336 to (87.61, -59.73, 107.55) mm, rotated rx 136.12 ry 0 rz -123.06 deg; joints [134.766, -14.816, 24.245, -99.379, 45.542, 122.148, 25, -236.939]
  MoveL 2337 to (78.4, -60.94, 113.79) mm, rotated rx 139.66 ry 0 rz -126.61 deg; joints [135.806, -13.456, 22.689, -98.866, 46.523, 118.118, 25, -233.387]
  MoveL 2338 to (77.11, -60.45, 114.92) mm, rotated rx 139.66 ry 0 rz -126.61 deg; joints [135.857, -13.413, 22.637, -98.843, 46.571, 118.096, 25, -233.387]
  MoveL 2339 to (76.61, -59.54, 115.72) mm, rotated rx 139.74 ry 0 rz -126.59 deg; joints [135.895, -13.335, 22.554, -98.826, 46.608, 117.998, 25, -233.407]
  MoveL 2340 to (76.35, -58.13, 116.62) mm, rotated rx 140.9 ry 0 rz -125.74 deg; joints [136.207, -12.944, 22.118, -98.691, 46.905, 116.709, 25, -234.265]
  MoveL 2341 to (75.78, -57.8, 117.15) mm, rotated rx 141.23 ry 0 rz -125.78 deg; joints [136.301, -12.815, 21.978, -98.652, 46.996, 116.348, 25, -234.221]
  MoveL 2342 to (75.2, -57.32, 117.75) mm, rotated rx 141.42 ry 0 rz -125.75 deg; joints [136.367, -12.724, 21.879, -98.625, 47.059, 116.134, 25, -234.254]
  MoveL 2343 to (74.91, -56.95, 118.12) mm, rotated rx 141.48 ry 0 rz -125.72 deg; joints [136.392, -12.684, 21.836, -98.615, 47.083, 116.065, 25, -234.282]
  MoveL 2344 to (73.34, -58.83, 118.2) mm, rotated rx 142.66 ry 0 rz -128.09 deg; joints [136.625, -12.266, 21.396, -98.527, 47.307, 114.813, 25, -231.915]
  MoveL 2345 to (70.71, -60.37, 119) mm, rotated rx 143.17 ry 0 rz -129.86 deg; joints [136.77, -12.06, 21.178, -98.473, 47.447, 114.257, 25, -230.142]
  MoveL 2346 to (70.79, -60.67, 118.79) mm, rotated rx 141.63 ry 0 rz -131.96 deg; joints [136.334, -12.451, 21.622, -98.65, 47.029, 115.949, 25, -228.042]
  MoveL 2347 to (71.84, -60.7, 118.15) mm, rotated rx 141.23 ry 0 rz -131.52 deg; joints [136.218, -12.611, 21.796, -98.698, 46.918, 116.396, 25, -228.476]
  MoveL 2348 to (73.06, -61.14, 117.19) mm, rotated rx 141.2 ry 0 rz -131.55 deg; joints [136.163, -12.653, 21.846, -98.722, 46.865, 116.446, 25, -228.454]
  MoveL 2349 to (73.58, -62.13, 116.35) mm, rotated rx 141.18 ry 0 rz -131.56 deg; joints [136.135, -12.715, 21.91, -98.732, 46.839, 116.478, 25, -228.436]
  MoveL 2350 to (73.11, -64.05, 115.6) mm, rotated rx 141.14 ry 0 rz -131.59 deg; joints [136.142, -12.818, 22.009, -98.726, 46.844, 116.506, 25, -228.408]
  MoveL 2351 to (71.05, -67.17, 115.11) mm, rotated rx 140.85 ry 0 rz -133.81 deg; joints [136.054, -12.931, 22.134, -98.763, 46.761, 116.835, 25, -226.185]
  MoveL 2352 to (70.39, -67.87, 115.11) mm, rotated rx 140.85 ry 0 rz -133.81 deg; joints [136.078, -12.963, 22.16, -98.751, 46.783, 116.823, 25, -226.185]
  MoveL 2353 to (69.96, -68.2, 115.17) mm, rotated rx 140.88 ry 0 rz -134.14 deg; joints [136.089, -12.948, 22.143, -98.746, 46.793, 116.782, 25, -225.864]
  MoveL 2354 to (66.65, -69.89, 116.11) mm, rotated rx 141.38 ry 0 rz -135.93 deg; joints [136.25, -12.761, 21.935, -98.678, 46.948, 116.22, 25, -224.073]
  MoveL 2355 to (66.68, -69.85, 116.12) mm, rotated rx 141.37 ry 0 rz -137.2 deg; joints [136.192, -12.694, 21.88, -98.707, 46.893, 116.262, 25, -222.797]
  MoveL 2356 to (66.19, -70.87, 115.79) mm, rotated rx 141.17 ry 0 rz -137.84 deg; joints [136.133, -12.773, 21.967, -98.731, 46.836, 116.487, 25, -222.158]
  MoveL 2357 to (65.72, -71.55, 115.64) mm, rotated rx 141.17 ry 0 rz -137.84 deg; joints [136.147, -12.807, 21.997, -98.723, 46.85, 116.478, 25, -222.158]
  MoveL 2358 to (64.95, -72.39, 115.55) mm, rotated rx 141.11 ry 0 rz -138.53 deg; joints [136.131, -12.827, 22.02, -98.73, 46.834, 116.54, 25, -221.475]
  MoveL 2359 to (60.06, -77.65, 114.76) mm, rotated rx 140.63 ry 0 rz -142.87 deg; joints [135.985, -13.006, 22.22, -98.794, 46.694, 117.082, 25, -217.132]
  MoveL 2360 to (60, -77.7, 114.78) mm, rotated rx 139.79 ry 0 rz -144.14 deg; joints [135.741, -13.194, 22.448, -98.906, 46.463, 118.021, 25, -215.856]
  MoveL 2361 to (60.17, -78.25, 114.31) mm, rotated rx 139.7 ry 0 rz -144.19 deg; joints [135.705, -13.249, 22.508, -98.922, 46.429, 118.128, 25, -215.811]
  MoveL 2362 to (60.29, -79.98, 113.05) mm, rotated rx 139.09 ry 0 rz -144.65 deg; joints [135.522, -13.5, 22.789, -99.006, 46.255, 118.817, 25, -215.353]
  MoveL 2363 to (60.74, -80.98, 112.08) mm, rotated rx 138.27 ry 0 rz -144.9 deg; joints [135.292, -13.787, 23.117, -99.117, 46.037, 119.744, 25, -215.104]
  MoveL 2364 to (61.07, -81.61, 111.43) mm, rotated rx 136.88 ry 0 rz -144.21 deg; joints [134.977, -14.281, 23.671, -99.273, 45.74, 121.288, 25, -215.789]
  MoveL 2365 to (63.9, -80.82, 110.4) mm, rotated rx 136.3 ry 0 rz -142.64 deg; joints [134.807, -14.502, 23.928, -99.362, 45.581, 121.953, 25, -217.363]
  MoveL 2366 to (63.79, -80.87, 110.43) mm, rotated rx 136.29 ry 0 rz -141.45 deg; joints [134.862, -14.58, 23.991, -99.331, 45.632, 121.934, 25, -218.555]
  MoveL 2367 to (64.44, -79.87, 110.78) mm, rotated rx 136.49 ry 0 rz -140.8 deg; joints [134.923, -14.505, 23.902, -99.298, 45.689, 121.699, 25, -219.201]
  MoveL 2368 to (65.17, -79.06, 110.94) mm, rotated rx 136.49 ry 0 rz -140.8 deg; joints [134.901, -14.462, 23.866, -99.311, 45.668, 121.712, 25, -219.201]
  MoveL 2369 to (66.37, -78.32, 110.76) mm, rotated rx 136.49 ry 0 rz -140.61 deg; joints [134.867, -14.436, 23.848, -99.33, 45.637, 121.733, 25, -219.387]
  MoveL 2370 to (68.83, -77.4, 109.9) mm, rotated rx 136.01 ry 0 rz -139.21 deg; joints [134.725, -14.62, 24.063, -99.406, 45.504, 122.29, 25, -220.794]
  MoveL 2371 to (70.19, -76.87, 109.4) mm, rotated rx 135.73 ry 0 rz -138.43 deg; joints [134.644, -14.725, 24.187, -99.45, 45.427, 122.612, 25, -221.569]
  MoveL 2372 to (70.42, -76.02, 109.85) mm, rotated rx 135.82 ry 0 rz -137.91 deg; joints [134.686, -14.686, 24.138, -99.427, 45.467, 122.501, 25, -222.092]
  MoveL 2373 to (71.95, -74.45, 109.94) mm, rotated rx 136.01 ry 0 rz -136.71 deg; joints [134.733, -14.624, 24.065, -99.401, 45.511, 122.282, 25, -223.288]
  MoveL 2374 to (72.52, -74.17, 109.75) mm, rotated rx 135.91 ry 0 rz -136.37 deg; joints [134.703, -14.663, 24.112, -99.418, 45.483, 122.401, 25, -223.63]
  MoveL 2375 to (73.43, -73.9, 109.33) mm, rotated rx 135.91 ry 0 rz -136.37 deg; joints [134.667, -14.654, 24.111, -99.438, 45.449, 122.422, 25, -223.63]
  MoveL 2376 to (79.17, -73.12, 105.8) mm, rotated rx 133.95 ry 0 rz -133.8 deg; joints [134.088, -15.384, 24.984, -99.768, 44.91, 124.711, 25, -226.2]
  MoveL 2377 to (82.04, -72.14, 104.27) mm, rotated rx 133.03 ry 0 rz -132.21 deg; joints [133.826, -15.726, 25.397, -99.928, 44.668, 125.796, 25, -227.794]
  MoveL 2378 to (82.67, -71.97, 103.89) mm, rotated rx 132.95 ry 0 rz -132.09 deg; joints [133.787, -15.751, 25.434, -99.952, 44.632, 125.897, 25, -227.905]
  MoveL 2379 to (85.46, -71.42, 102) mm, rotated rx 131.86 ry 0 rz -130.85 deg; joints [133.467, -16.144, 25.922, -100.158, 44.338, 127.205, 25, -229.152]
  MoveL 2380 to (86.69, -71.65, 100.79) mm, rotated rx 131.86 ry 0 rz -130.85 deg; joints [133.411, -16.17, 25.965, -100.194, 44.287, 127.243, 25, -229.152]
  MoveL 2381 to (87.19, -72.43, 99.79) mm, rotated rx 131.79 ry 0 rz -130.85 deg; joints [133.368, -16.238, 26.046, -100.223, 44.248, 127.345, 25, -229.154]
  MoveL 2382 to (87.39, -73.34, 98.95) mm, rotated rx 131.37 ry 0 rz -131.13 deg; joints [133.241, -16.388, 26.237, -100.309, 44.131, 127.855, 25, -228.872]
  MoveL 2383 to (88.05, -74.11, 97.79) mm, rotated rx 130.47 ry 0 rz -131.32 deg; joints [132.984, -16.672, 26.606, -100.487, 43.898, 128.933, 25, -228.675]
  Set speed (16.7 mm/s)
  MoveL 2384 to (99.47, -84.16, 110.77) mm, rotated rx 130.47 ry 0 rz -131.32 deg; joints [132.76, -16.976, 26.19, -99.823, 43.553, 127.963, 25, -228.675]
  Set speed (1000.0 mm/s)
  MoveL 2385 to (96.52, -88.4, 110.08) mm, rotated rx 130.58 ry 0 rz -131.62 deg; joints [132.875, -17.127, 26.302, -99.746, 43.659, 127.772, 25, -228.375]
  Set speed (5.0 mm/s)
  MoveL 2386 to (85.16, -78.31, 97.07) mm, rotated rx 130.58 ry 0 rz -131.62 deg; joints [133.099, -16.824, 26.721, -100.408, 44.003, 128.742, 25, -228.375]
  Set speed (16.7 mm/s)
  MoveL 2387 to (84.42, -78.42, 97.62) mm, rotated rx 130.86 ry 0 rz -131.91 deg; joints [133.182, -16.726, 26.596, -100.351, 44.079, 128.407, 25, -228.094]
  MoveL 2388 to (84.43, -78.36, 97.65) mm, rotated rx 130.44 ry 0 rz -134.09 deg; joints [132.972, -16.687, 26.625, -100.495, 43.887, 128.976, 25, -225.906]
  MoveL 2389 to (85.4, -79.89, 95.56) mm, rotated rx 129.41 ry 0 rz -134.3 deg; joints [132.659, -17.048, 27.096, -100.722, 43.604, 130.245, 25, -225.696]
  MoveL 2390 to (86.47, -80.7, 93.9) mm, rotated rx 128.4 ry 0 rz -134.24 deg; joints [132.364, -17.38, 27.538, -100.945, 43.34, 131.492, 25, -225.765]
  MoveL 2391 to (86.78, -81.13, 93.24) mm, rotated rx 128.3 ry 0 rz -134.26 deg; joints [132.321, -17.43, 27.604, -100.978, 43.302, 131.622, 25, -225.743]
  MoveL 2392 to (87.3, -83.14, 90.96) mm, rotated rx 127.39 ry 0 rz -134.71 deg; joints [132.034, -17.758, 28.047, -101.207, 43.046, 132.784, 25, -225.29]
  MoveL 2393 to (87.98, -84.68, 88.86) mm, rotated rx 126.27 ry 0 rz -135.05 deg; joints [131.699, -18.117, 28.546, -101.484, 42.751, 134.197, 25, -224.954]
  MoveL 2394 to (88.07, -85.09, 88.38) mm, rotated rx 126.27 ry 0 rz -135.05 deg; joints [131.69, -18.142, 28.574, -101.492, 42.743, 134.206, 25, -224.954]
  MoveL 2395 to (87.89, -86.33, 87.35) mm, rotated rx 126.12 ry 0 rz -135.14 deg; joints [131.644, -18.242, 28.696, -101.533, 42.702, 134.397, 25, -224.858]
  MoveL 2396 to (86.28, -89.88, 85.35) mm, rotated rx 125.37 ry 0 rz -136.54 deg; joints [131.42, -18.521, 29.076, -101.73, 42.507, 135.357, 25, -223.465]
  MoveL 2397 to (85.37, -91.08, 85.01) mm, rotated rx 125.37 ry 0 rz -136.54 deg; joints [131.447, -18.586, 29.132, -101.709, 42.531, 135.335, 25, -223.465]
  MoveL 2398 to (84.57, -91.73, 85.12) mm, rotated rx 125.38 ry 0 rz -136.7 deg; joints [131.468, -18.605, 29.143, -101.692, 42.55, 135.312, 25, -223.304]
  MoveL 2399 to (83.35, -92.49, 85.48) mm, rotated rx 125.55 ry 0 rz -137.36 deg; joints [131.521, -18.548, 29.062, -101.646, 42.596, 135.088, 25, -222.643]
  MoveL 2400 to (83.33, -92.48, 85.48) mm, rotated rx 125.31 ry 0 rz -138.57 deg; joints [131.396, -18.516, 29.081, -101.75, 42.486, 135.446, 25, -221.434]
  MoveL 2401 to (82.96, -93.63, 84.59) mm, rotated rx 124.89 ry 0 rz -139.05 deg; joints [131.27, -18.649, 29.272, -101.863, 42.377, 135.98, 25, -220.955]
  MoveL 2402 to (82.93, -93.6, 84.67) mm, rotated rx 124.13 ry 0 rz -139.76 deg; joints [131.051, -18.783, 29.505, -102.059, 42.187, 136.956, 25, -220.245]
  MoveL 2403 to (83.7, -94.23, 83.21) mm, rotated rx 123.45 ry 0 rz -139.67 deg; joints [130.845, -18.997, 29.819, -102.253, 42.01, 137.845, 25, -220.334]
  MoveL 2404 to (84.01, -94.85, 82.19) mm, rotated rx 123.45 ry 0 rz -139.67 deg; joints [130.819, -19.034, 29.87, -102.278, 41.988, 137.872, 25, -220.334]
  MoveL 2405 to (83.95, -95.66, 81.3) mm, rotated rx 123.29 ry 0 rz -139.75 deg; joints [130.765, -19.115, 29.979, -102.332, 41.942, 138.09, 25, -220.255]
  MoveL 2406 to (83.68, -96.53, 80.53) mm, rotated rx 122.97 ry 0 rz -140.06 deg; joints [130.667, -19.219, 30.132, -102.427, 41.859, 138.517, 25, -219.937]
  MoveL 2407 to (83.66, -96.49, 80.59) mm, rotated rx 121.55 ry 0 rz -139.79 deg; joints [130.346, -19.581, 30.664, -102.751, 41.588, 140.286, 25, -220.208]
  MoveL 2408 to (84.44, -96.18, 80.17) mm, rotated rx 121.35 ry 0 rz -139.42 deg; joints [130.287, -19.641, 30.756, -102.812, 41.538, 140.548, 25, -220.576]
  MoveL 2409 to (84.87, -96, 79.93) mm, rotated rx 121.24 ry 0 rz -139.23 deg; joints [130.254, -19.674, 30.806, -102.846, 41.511, 140.692, 25, -220.774]
  MoveL 2410 to (89.89, -94.29, 76.4) mm, rotated rx 119.67 ry 0 rz -137.08 deg; joints [129.778, -20.14, 31.539, -103.356, 41.117, 142.826, 25, -222.921]
  MoveL 2411 to (90.53, -94.13, 75.84) mm, rotated rx 119.54 ry 0 rz -136.96 deg; joints [129.725, -20.171, 31.6, -103.412, 41.073, 143.011, 25, -223.039]
  MoveL 2412 to (91.88, -94.11, 74.2) mm, rotated rx 119.02 ry 0 rz -136.67 deg; joints [129.547, -20.322, 31.856, -103.612, 40.928, 143.754, 25, -223.333]
  MoveL 2413 to (85.22, -103.24, 69.89) mm, rotated rx 117.88 ry 0 rz -139.45 deg; joints [129.275, -20.862, 32.583, -103.952, 40.714, 145.263, 25, -220.547]
  MoveL 2414 to (84.46, -103.07, 71.07) mm, rotated rx 118.39 ry 0 rz -139.65 deg; joints [129.426, -20.72, 32.347, -103.774, 40.835, 144.564, 25, -220.348]
  MoveL 2415 to (82.9, -103.3, 72.55) mm, rotated rx 119.34 ry 0 rz -140.53 deg; joints [129.675, -20.441, 31.914, -103.485, 41.036, 143.292, 25, -219.473]
  MoveL 2416 to (82.42, -103.29, 73.11) mm, rotated rx 119.4 ry 0 rz -140.56 deg; joints [129.711, -20.424, 31.878, -103.446, 41.066, 143.194, 25, -219.445]
  MoveL 2417 to (81.9, -103.11, 73.93) mm, rotated rx 119.62 ry 0 rz -140.62 deg; joints [129.789, -20.358, 31.766, -103.36, 41.13, 142.884, 25, -219.378]
  MoveL 2418 to (82.03, -103.07, 73.83) mm, rotated rx 120.25 ry 0 rz -141.34 deg; joints [129.892, -20.148, 31.489, -103.238, 41.213, 142.116, 25, -218.66]
  MoveL 2419 to (79.28, -104.67, 74.61) mm, rotated rx 120.59 ry 0 rz -142.74 deg; joints [129.993, -20.046, 31.329, -103.128, 41.296, 141.655, 25, -217.256]
  MoveL 2420 to (78.73, -104.93, 74.82) mm, rotated rx 120.59 ry 0 rz -142.74 deg; joints [130.014, -20.062, 31.336, -103.108, 41.313, 141.634, 25, -217.256]
  MoveL 2421 to (77.17, -105.18, 76.07) mm, rotated rx 120.67 ry 0 rz -142.89 deg; joints [130.094, -20.049, 31.282, -103.028, 41.38, 141.472, 25, -217.108]
  MoveL 2422 to (75.93, -104.81, 77.8) mm, rotated rx 121.44 ry 0 rz -143.24 deg; joints [130.327, -19.817, 30.922, -102.784, 41.575, 140.433, 25, -216.763]
  MoveL 2423 to (75.93, -104.84, 77.76) mm, rotated rx 122.01 ry 0 rz -144.02 deg; joints [130.419, -19.617, 30.667, -102.684, 41.651, 139.75, 25, -215.983]
  MoveL 2424 to (72.76, -106.49, 78.55) mm, rotated rx 122.36 ry 0 rz -145.62 deg; joints [130.523, -19.507, 30.502, -102.578, 41.738, 139.284, 25, -214.382]
  MoveL 2425 to (71.88, -107.61, 77.86) mm, rotated rx 121.96 ry 0 rz -147.05 deg; joints [130.361, -19.554, 30.628, -102.735, 41.601, 139.853, 25, -212.946]
  Set speed (16.7 mm/s)
  MoveL 2426 to (81.1, -121.85, 88.44) mm, rotated rx 121.96 ry 0 rz -147.05 deg; joints [130.04, -19.947, 30.315, -102.089, 41.141, 138.912, 25, -212.946]
  Set speed (1000.0 mm/s)
  MoveL 2427 to (76.27, -124.33, 89.28) mm, rotated rx 121.88 ry 0 rz -147.82 deg; joints [130.131, -20.071, 30.401, -102.009, 41.22, 138.909, 25, -212.177]
  Set speed (5.0 mm/s)
  MoveL 2428 to (67.23, -109.95, 78.71) mm, rotated rx 121.88 ry 0 rz -147.82 deg; joints [130.452, -19.676, 30.713, -102.655, 41.679, 139.85, 25, -212.177]
  Set speed (16.7 mm/s)
  MoveL 2429 to (66.34, -109.64, 79.86) mm, rotated rx 122.41 ry 0 rz -148.09 deg; joints [130.61, -19.515, 30.47, -102.496, 41.813, 139.153, 25, -211.91]
  MoveL 2430 to (66.4, -109.69, 79.77) mm, rotated rx 122.7 ry 0 rz -149.89 deg; joints [130.576, -19.298, 30.258, -102.517, 41.782, 138.881, 25, -210.111]
  MoveL 2431 to (65.6, -110.87, 78.81) mm, rotated rx 122.26 ry 0 rz -150.47 deg; joints [130.443, -19.432, 30.461, -102.65, 41.669, 139.464, 25, -209.53]
  MoveL 2432 to (65.51, -110.88, 78.88) mm, rotated rx 120.69 ry 0 rz -150.23 deg; joints [130.087, -19.825, 31.048, -103.02, 41.372, 141.433, 25, -209.771]
  MoveL 2433 to (66.11, -110.73, 78.59) mm, rotated rx 120.67 ry 0 rz -150.16 deg; joints [130.062, -19.823, 31.058, -103.045, 41.35, 141.486, 25, -209.836]
  MoveL 2434 to (67.55, -110.49, 77.7) mm, rotated rx 120.26 ry 0 rz -149.55 deg; joints [129.941, -19.943, 31.246, -103.174, 41.251, 142.03, 25, -210.455]
  Set speed (16.7 mm/s)
  MoveL 2435 to (76.3, -125.38, 87.78) mm, rotated rx 120.26 ry 0 rz -149.55 deg; joints [129.602, -20.352, 30.955, -102.538, 40.77, 141.101, 25, -210.455]
  Set speed (1000.0 mm/s)
  MoveL 2436 to (81.3, -122.05, 87.96) mm, rotated rx 120.21 ry 0 rz -146.86 deg; joints [129.616, -20.393, 30.991, -102.527, 40.783, 141.145, 25, -213.141]
  Set speed (5.0 mm/s)
  MoveL 2437 to (71.85, -107.58, 77.9) mm, rotated rx 120.21 ry 0 rz -146.86 deg; joints [129.956, -19.983, 31.282, -103.163, 41.264, 142.073, 25, -213.141]
  Set speed (16.7 mm/s)
  MoveL 2438 to (74.32, -106.44, 77.17) mm, rotated rx 119.88 ry 0 rz -145.64 deg; joints [129.858, -20.082, 31.436, -103.268, 41.183, 142.517, 25, -214.357]
  MoveL 2439 to (76.08, -106.16, 75.83) mm, rotated rx 119.88 ry 0 rz -145.64 deg; joints [129.781, -20.058, 31.45, -103.346, 41.118, 142.6, 25, -214.357]
  MoveL 2440 to (76.49, -107.22, 73.91) mm, rotated rx 119.88 ry 0 rz -145.64 deg; joints [129.733, -20.119, 31.541, -103.4, 41.079, 142.659, 25, -214.357]
  MoveL 2441 to (76.36, -107.61, 73.48) mm, rotated rx 119.69 ry 0 rz -145.79 deg; joints [129.675, -20.175, 31.63, -103.465, 41.032, 142.922, 25, -214.211]
  MoveL 2442 to (74.64, -110.62, 70.67) mm, rotated rx 118.61 ry 0 rz -147.01 deg; joints [129.35, -20.501, 32.154, -103.839, 40.769, 144.412, 25, -212.988]
  MoveL 2443 to (74.55, -110.64, 70.76) mm, rotated rx 117.18 ry 0 rz -146.89 deg; joints [129.027, -20.825, 32.684, -104.227, 40.512, 146.259, 25, -213.114]
  MoveL 2444 to (75.37, -110.41, 70.28) mm, rotated rx 116.97 ry 0 rz -146.53 deg; joints [128.964, -20.884, 32.784, -104.304, 40.462, 146.556, 25, -213.467]
  MoveL 2445 to (75.8, -110.29, 70) mm, rotated rx 116.87 ry 0 rz -146.38 deg; joints [128.931, -20.909, 32.83, -104.344, 40.436, 146.698, 25, -213.617]
  MoveL 2446 to (80.22, -109.48, 66.24) mm, rotated rx 115.34 ry 0 rz -144.73 deg; joints [128.469, -21.311, 33.544, -104.932, 40.078, 148.87, 25, -215.266]
  MoveL 2447 to (81.82, -108.86, 65.3) mm, rotated rx 114.8 ry 0 rz -143.83 deg; joints [128.33, -21.462, 33.796, -105.119, 39.973, 149.618, 25, -216.165]
  MoveL 2448 to (82.54, -108.68, 64.7) mm, rotated rx 114.8 ry 0 rz -143.83 deg; joints [128.298, -21.449, 33.802, -105.158, 39.948, 149.659, 25, -216.165]
  MoveL 2449 to (82.97, -108.65, 64.19) mm, rotated rx 114.69 ry 0 rz -143.75 deg; joints [128.255, -21.476, 33.859, -105.215, 39.915, 149.831, 25, -216.251]
  MoveL 2450 to (84.56, -108.68, 62.03) mm, rotated rx 113.77 ry 0 rz -143.21 deg; joints [127.987, -21.709, 34.288, -105.584, 39.715, 151.158, 25, -216.786]
  MoveL 2451 to (85.24, -109.09, 60.34) mm, rotated rx 112.69 ry 0 rz -142.72 deg; joints [127.718, -21.99, 34.781, -105.975, 39.52, 152.673, 25, -217.284]
  MoveL 2452 to (86.29, -108.63, 59.69) mm, rotated rx 112.41 ry 0 rz -142.24 deg; joints [127.64, -22.056, 34.909, -106.089, 39.464, 153.071, 25, -217.755]
  MoveL 2453 to (86.91, -108.41, 59.18) mm, rotated rx 112.41 ry 0 rz -142.24 deg; joints [127.612, -22.042, 34.912, -106.125, 39.443, 153.11, 25, -217.755]
  MoveL 2454 to (87.75, -108.62, 57.54) mm, rotated rx 112.41 ry 0 rz -142.24 deg; joints [127.557, -22.055, 34.964, -106.202, 39.402, 153.193, 25, -217.755]
  MoveL 2455 to (87.87, -108.87, 56.87) mm, rotated rx 112.14 ry 0 rz -142.27 deg; joints [127.477, -22.12, 35.094, -106.321, 39.346, 153.603, 25, -217.73]
  MoveL 2456 to (87.86, -111.36, 51.85) mm, rotated rx 110.24 ry 0 rz -142.86 deg; joints [126.93, -22.56, 35.992, -107.174, 38.967, 156.435, 25, -217.137]
  MoveL 2457 to (87.86, -111.88, 50.72) mm, rotated rx 109.75 ry 0 rz -143 deg; joints [126.793, -22.665, 36.217, -107.397, 38.875, 157.174, 25, -217.001]
  MoveL 2458 to (87.76, -112.25, 50.06) mm, rotated rx 109.75 ry 0 rz -143 deg; joints [126.784, -22.689, 36.252, -107.414, 38.871, 157.193, 25, -217.001]
  MoveL 2459 to (84.83, -117.8, 41.63) mm, rotated rx 106.56 ry 0 rz -144.87 deg; joints [125.917, -23.376, 37.771, -108.943, 38.33, 162.068, 25, -215.128]
  MoveL 2460 to (84.28, -118.46, 40.86) mm, rotated rx 106.56 ry 0 rz -144.87 deg; joints [125.919, -23.423, 37.825, -108.95, 38.335, 162.076, 25, -215.128]
  MoveL 2461 to (83.55, -119.18, 40.28) mm, rotated rx 106.33 ry 0 rz -145.28 deg; joints [125.857, -23.465, 37.93, -109.066, 38.298, 162.434, 25, -214.722]
  MoveL 2462 to (74.71, -125.93, 36.97) mm, rotated rx 105.08 ry 0 rz -149.61 deg; joints [125.519, -23.694, 38.514, -109.714, 38.109, 164.407, 25, -210.394]
  MoveL 2463 to (72.85, -127.36, 35.78) mm, rotated rx 104.54 ry 0 rz -150.69 deg; joints [125.372, -23.764, 38.739, -110.001, 38.027, 165.255, 25, -209.311]
  MoveL 2464 to (72.33, -127.72, 35.56) mm, rotated rx 104.54 ry 0 rz -150.69 deg; joints [125.382, -23.794, 38.766, -109.99, 38.035, 165.245, 25, -209.311]
  MoveL 2465 to (71.7, -128.11, 35.4) mm, rotated rx 104.48 ry 0 rz -150.98 deg; joints [125.366, -23.804, 38.794, -110.023, 38.027, 165.343, 25, -209.022]
  MoveL 2466 to (69.43, -129.62, 34.29) mm, rotated rx 104.01 ry 0 rz -152.19 deg; joints [125.235, -23.863, 38.996, -110.284, 37.957, 166.109, 25, -207.809]
  MoveL 2467 to (70.26, -129.64, 32.62) mm, rotated rx 102.47 ry 0 rz -152.52 deg; joints [124.849, -24.008, 39.567, -111.068, 37.759, 168.509, 25, -207.483]
  MoveL 2468 to (70.31, -129.74, 32.11) mm, rotated rx 102.27 ry 0 rz -152.52 deg; joints [124.798, -24.038, 39.658, -111.178, 37.736, 168.83, 25, -207.484]
  MoveL 2469 to (69.83, -130.42, 30.36) mm, rotated rx 102.27 ry 0 rz -152.52 deg; joints [124.779, -24.091, 39.745, -111.233, 37.731, 168.893, 25, -207.484]
  MoveL 2470 to (67.3, -132.41, 27.29) mm, rotated rx 101.08 ry 0 rz -153.74 deg; joints [124.481, -24.258, 40.282, -111.897, 37.6, 170.814, 25, -206.264]
  MoveL 2471 to (65.83, -133.29, 26.58) mm, rotated rx 101.08 ry 0 rz -153.74 deg; joints [124.507, -24.34, 40.358, -111.87, 37.621, 170.79, 25, -206.264]
  MoveL 2472 to (64.21, -134, 26.97) mm, rotated rx 101.08 ry 0 rz -153.87 deg; joints [124.548, -24.398, 40.386, -111.803, 37.647, 170.722, 25, -206.133]
  MoveL 2473 to (63.32, -134.29, 27.58) mm, rotated rx 101.32 ry 0 rz -154.23 deg; joints [124.606, -24.366, 40.28, -111.672, 37.671, 170.343, 25, -205.773]
  Set speed (1000.0 mm/s)
  MoveL 2474 to (63.32, -134.29, 27.58) mm, rotated rx 101.32 ry 0 rz -154.23 deg; joints [124.606, -24.366, 40.28, -111.672, 37.671, 170.343, 25, -205.773]
  MoveL 2475 to (105.95, -222.6, 47.2) mm, rotated rx 101.32 ry 0 rz -154.23 deg; joints [121.756, -27.097, 39.926, -109.735, 33.996, 167.083, 25, -205.773]
  Call onMillingEarth_Retract
  Call onMillingEarth_Finish
